# B&R Automation Studio project Soiled_PLC (part 8)

#### pr.st - Implementation code
```iecst
(********************************************************************
 * COPYRIGHT --
 ********************************************************************
 * Program: pr
 * File: pr.st
 * Author: treamsbottom
 * Created: July 16, 2015
 ********************************************************************
 * Implementation of program pr
 ********************************************************************)

PROGRAM _INIT
//Configuration
mySeq						:= 23;	//Sequence number
myIO						:= 11;
myZone						:= 0;
myRelLine					:= 31;
myBag						:= 243; //Buffer Bag
bufferSettleTime			:= 300;

myOutBag 					:= Line[myRelLine].LastBag;
END_PROGRAM

PROGRAM _CYCLIC
//Inputs
i_bagAtBuffer				:= X[myIO].X01;

i_bagAtBufferOut 		:= FALSE; // Any Single bag buffer out IO.
i_bufferOutOpen			:= FALSE;

o_openBuffer	:= FALSE;

IF (myBag = 0) THEN
	Alarm[mySeq].Bag	:= mySeq + 10000;
ELSE
	Alarm[mySeq].Bag	:= myBag;
END_IF;

Alarm[mySeq].Name 		:= 0;
Alarm[mySeq].Beacon		:= TRUE;
Alarm[mySeq].Extra		:= 0;
Alarm[mySeq].Time		:= 3000;

//Setup Sequence
step := D[900 + mySeq];
//Setup Pulse contact
pls := (step <> lastStep);
lastStep := step;

//Sequence
IF (step = 0) THEN
	//Disabled
END_IF;

//Bag Settled at buffer
ton_10ms_SettledBuffer(IN:= i_bagAtBuffer, PT:= bufferSettleTime);
IF (step = 1) THEN
	IF ton_10ms_SettledBuffer.Q AND NOT Std.HaltSysZone[myZone]THEN
		IF Line[myRelLine].Clear AND NOT i_bagAtBufferOut AND NOT i_bufferOutOpen AND NOT Line[myRelLine].Trip THEN
			IF (myBag = 0) THEN
				C[myRelLine] := 0;
				D[900 + mySeq] := 2;
			ELSIF (Bag[myBag].Cat > 0) AND (Bag[myOutBag].Cat = 0) THEN
				C[myRelLine] := 0;
				D[900 + mySeq] := 2;
			ELSIF (Bag[myBag].Cat = 0) THEN
				Alarm[mySeq].Name := ALM_BAG_DATA_ERROR;
				Alarm[mySeq].Time := 0;
			ELSIF (Bag[myOutBag].Cat > 0) THEN
				Alarm[mySeq].Name := ALM_BAG_DATA_ERROR;
				Alarm[mySeq].Bag := myOutBag;
				Alarm[mySeq].Time := 0;
			END_IF;
		ELSIF Line[myRelLine].Trip THEN
			Alarm[mySeq].Name := ALM_SWITCH_FAULT; //Trip is stuck on
			Alarm[mySeq].Time := 500;
		END_IF;
	ELSIF (myBag > 0) AND (Bag[myBag].Cat > 0) THEN
		Alarm[mySeq].Name := ALM_BAG_NOT_SETTLED;
	END_IF;
END_IF;

IF (step = 2) THEN
	dataValid := ((myBag = 0) OR ((Bag[myBag].Cat > 0) AND (Bag[myOutBag].Cat = 0)));
	o_openBuffer :=  dataValid;
	IF dataValid THEN
		IF Line[myRelLine].Trip THEN
			IF (myBag > 0) THEN
				Bag[myOutBag] := Bag[myBag];
				Bag[myBag]  := Bag[0];
			END_IF;
			D[900 + mySeq] := 1;
		END_IF;
		Alarm[mySeq].Name := ALM_BAG_NOT_RELEASED;
	ELSIF (myBag > 0) THEN
		IF (Bag[myBag].Cat = 0) THEN
			Alarm[mySeq].Name := ALM_BAG_DATA_ERROR;
			Alarm[mySeq].Time := 0;
		ELSIF (Bag[myOutBag].Cat > 0) THEN
			Alarm[mySeq].Name := ALM_BAG_DATA_ERROR;
			Alarm[mySeq].Bag := myOutBag;
			Alarm[mySeq].Time := 0;
		END_IF;
	END_IF;
END_IF;

//-----------------------------------
//PLC Outputs - adjust TO suit system
//-----------------------------------

Y[myIO].Y01 := o_openBuffer;

//Alarms
timerAlarm(IN := NOT pls AND (Alarm[mySeq].Name > 0),PT:= Alarm[mySeq].Time);

Alarm[mySeq].On 	:= timerAlarm.Q;
Alarm[mySeq].ET 	:= timerAlarm.ET;

END_PROGRAM
```

### Program Logical/Sequences/10ms/zzForceO (IEC)

#### zzforceo.ab
```automation-basic
;----------------------------
;Output forcing from Graphics
;----------------------------

;Version 1.00 02/09/2006 D.J. First Issue
;Version 2.00 20/11/2009 D.J. Changed to 8 I/O inputs per card

PROGRAM _INIT

;Clear force registers

D[380] = 0
D[381] = 0
D[382] = 0
D[383] = 0
D[384] = 0
D[385] = 0
D[386] = 0
D[386] = 0
D[387] = 0
D[388] = 0
D[389] = 0
D[390] = 0
D[391] = 0
D[392] = 0
D[393] = 0
D[394] = 0
D[395] = 0
D[396] = 0
D[396] = 0
D[397] = 0
D[398] = 0
D[399] = 0

;Clear force disable
memset(ADR(YForceDisable),0, SIZEOF(YForceDisable))

END_PROGRAM

PROGRAM _CYCLIC

LOOP Force = 1 TO 4 DO

	n = ((Force - 1) * 5)

	myForceCard 	= D[380 + n]
	myForceState 	= D[383 + n]
	myForceValue 	= D[384 + n]

	IF (myForceCard > Std.MaxIO) THEN
		myForceCard = 0
	ENDIF

	YForce.Y01 		= BIT_TST(myForceState,0)
	YForce.Y02 		= BIT_TST(myForceState,1)
	YForce.Y03 		= BIT_TST(myForceState,2)
	YForce.Y04 		= BIT_TST(myForceState,3)
	YForce.Y05 		= BIT_TST(myForceState,4)
	YForce.Y06 		= BIT_TST(myForceState,5)
	YForce.Y07 		= BIT_TST(myForceState,6)
	YForce.Y08 		= BIT_TST(myForceState,7)
	YForce.Y09 		= BIT_TST(myForceState,8)
	YForce.Y10 		= BIT_TST(myForceState,9)
	YForce.Y11 		= BIT_TST(myForceState,10)
	YForce.Y12 		= BIT_TST(myForceState,11)
	YForce.Y13 		= BIT_TST(myForceState,12)
	YForce.Y14 		= BIT_TST(myForceState,13)
	YForce.Y15 		= BIT_TST(myForceState,14)
	YForce.Y16 		= BIT_TST(myForceState,15)

	YForceVal.Y01 	= BIT_TST(myForceValue,0)
	YForceVal.Y02 	= BIT_TST(myForceValue,1)
	YForceVal.Y03 	= BIT_TST(myForceValue,2)
	YForceVal.Y04 	= BIT_TST(myForceValue,3)
	YForceVal.Y05 	= BIT_TST(myForceValue,4)
	YForceVal.Y06 	= BIT_TST(myForceValue,5)
	YForceVal.Y07 	= BIT_TST(myForceValue,6)
	YForceVal.Y08 	= BIT_TST(myForceValue,7)
	YForceVal.Y09 	= BIT_TST(myForceValue,8)
	YForceVal.Y10 	= BIT_TST(myForceValue,9)
	YForceVal.Y11 	= BIT_TST(myForceValue,10)
	YForceVal.Y12 	= BIT_TST(myForceValue,11)
	YForceVal.Y13 	= BIT_TST(myForceValue,12)
	YForceVal.Y14 	= BIT_TST(myForceValue,13)
	YForceVal.Y15 	= BIT_TST(myForceValue,14)
	YForceVal.Y16 	= BIT_TST(myForceValue,15)

	Y[myForceCard].Y01 = (Y[myForceCard].Y01 AND NOT YForce.Y01) OR (YForce.Y01 AND YForceVal.Y01)
	Y[myForceCard].Y02 = (Y[myForceCard].Y02 AND NOT YForce.Y02) OR (YForce.Y02 AND YForceVal.Y02)
	Y[myForceCard].Y03 = (Y[myForceCard].Y03 AND NOT YForce.Y03) OR (YForce.Y03 AND YForceVal.Y03)
	Y[myForceCard].Y04 = (Y[myForceCard].Y04 AND NOT YForce.Y04) OR (YForce.Y04 AND YForceVal.Y04)
	Y[myForceCard].Y05 = (Y[myForceCard].Y05 AND NOT YForce.Y05) OR (YForce.Y05 AND YForceVal.Y05)
	Y[myForceCard].Y06 = (Y[myForceCard].Y06 AND NOT YForce.Y06) OR (YForce.Y06 AND YForceVal.Y06)
	Y[myForceCard].Y07 = (Y[myForceCard].Y07 AND NOT YForce.Y07) OR (YForce.Y07 AND YForceVal.Y07)
	Y[myForceCard].Y08 = (Y[myForceCard].Y08 AND NOT YForce.Y08) OR (YForce.Y08 AND YForceVal.Y08)
	Y[myForceCard].Y09 = (Y[myForceCard].Y09 AND NOT YForce.Y09) OR (YForce.Y09 AND YForceVal.Y09)
	Y[myForceCard].Y10 = (Y[myForceCard].Y10 AND NOT YForce.Y10) OR (YForce.Y10 AND YForceVal.Y10)
	Y[myForceCard].Y11 = (Y[myForceCard].Y11 AND NOT YForce.Y11) OR (YForce.Y11 AND YForceVal.Y11)
	Y[myForceCard].Y12 = (Y[myForceCard].Y12 AND NOT YForce.Y12) OR (YForce.Y12 AND YForceVal.Y12)
	Y[myForceCard].Y13 = (Y[myForceCard].Y13 AND NOT YForce.Y13) OR (YForce.Y13 AND YForceVal.Y13)
	Y[myForceCard].Y14 = (Y[myForceCard].Y14 AND NOT YForce.Y14) OR (YForce.Y14 AND YForceVal.Y14)
	Y[myForceCard].Y15 = (Y[myForceCard].Y15 AND NOT YForce.Y15) OR (YForce.Y15 AND YForceVal.Y15)
	Y[myForceCard].Y16 = (Y[myForceCard].Y16 AND NOT YForce.Y16) OR (YForce.Y16 AND YForceVal.Y16)

ENDLOOP

END_PROGRAM
```

### Program Logical/Sequences/10ms/zzStnSer (IEC, version 3.00.1)

#### zzstnser.var
```iecst
VAR
	MixProgTyp : BOOL;
	BatchFound : BOOL;
	MixCusts : BOOL;
	MixProgs : BOOL;
	MatchCust : BOOL;
	MatchBags : BOOL;
	MatchProgType : BOOL;
	MatchProg : BOOL;
	MatchCat : BOOL;
	StartPurge : BOOL;
	MixCats : BOOL;
	BankValid : BOOL;
	LineValid : BOOL;
	BagInList : ARRAY[0..30] OF BOOL;
	StartPurgeET : UDINT;
	BagNum : UINT;
	BagWgt : UINT;
	Index : UINT;
	PurgeBagsQty : UINT;
	StnNum : UINT;
	BatchCount : UINT;
	s : UINT;
	BatchWeight : UINT;
	myBag : UINT;
	r : UINT;
	MaxReverseWeight : UINT;
END_VAR
VAR RETAIN
	LineSearchManual : UINT;
END_VAR
VAR
	NumberOfPurgeBags : UINT;
	x : UINT;
END_VAR
VAR RETAIN
	SearchLine : UINT;
END_VAR
VAR
	Bank : UINT;
	Choice : UINT;
	EndofBagArray : UINT;
	PurgeBatchSize : UINT;
	MaxBatchWieght : UINT;
END_VAR
VAR RETAIN
	n : UINT;
END_VAR
VAR
	t : UINT;
	myBag_x : UINT;
	myBag_n : UINT;
END_VAR
VAR RETAIN
	SearchFound : UINT;
END_VAR
VAR
	LineSearch : ARRAY[0..4] OF UINT;
	SearchBagArray : ARRAY[0..30] OF UINT;
	PurgeBags : ARRAY[0..30] OF UINT;
	PurgeBagsInWgtOrder : ARRAY[0..30] OF UINT;
	PurgeOn : UINT;
	StatusReg : ARRAY[0..1] OF UDINT;
	SearchIndex : USINT;
	ReSearch : BOOL;
	MisMatchedLoad : BOOL;
	y : INT;
	Break : BOOL;
	StnCat : UDINT;
	GetStn : UINT;
	TestTim : BOOL;
	myStartStop : UINT;
	b : UINT;
	TON_Purge : ARRAY[0..4] OF TON_10ms;
	myBatchWgt : UDINT;
	test : UDINT;
	TEST : BOOL;
END_VAR
```

#### zzstnser.ab
```automation-basic
;-----------------------------------------------------
;Sorting Station Search Routine - No changes required!
;-----------------------------------------------------

;----------------------------------------
;Version 1.00 19/12/2005 First Issue D.J.
;Version 2.00 03/11/2010 Revised D.J.
;Version 3.00 19/07/2016 TR... Fix bug so multiple banks can release whilst purging..
;----------------------------------------

PROGRAM _CYCLIC

;Only one Bank / Loading VC can search in a given scan.

myStartStop			= 100 ; Start of Start Stops

IF myStartStop >= 100 THEN
	myStartStop = myStartStop + 7600
ENDIF

Bank = Bank + 1
IF (Bank > Std.MaxStationBanks) THEN
	Bank = 1
ENDIF
;Clear arrays
LOOP n = 0 TO Std.MaxWeighstations DO
	BagInList[n] = FALSE
	SearchBagArray[n] = 0
ENDLOOP

;Clear Array
LOOP b = 1 TO 4 DO
	Std.StnsToPurge[b] = FALSE
	LOOP n = 1 TO Ldg[b].NoStations DO
		x = Ldg[b].Stations[n]
		IF Stn[x].Purge THEN
			Std.StnsToPurge[b] = TRUE
		ENDIF
	ENDLOOP
	TON_Purge[b].IN = Std.StnsToPurge[b]
	TON_Purge[b].PT = 100
	TON_Purge[b] FUB TON_10ms()
	//TON_10ms(Std.StnsToPurge,100,StartPurge,StartPurgeET) ; use a timer to wait for all purge events to be recieved from trackview
ENDLOOP

MixCats			= (D[369] > 0)
MixCusts		= (D[366] > 0)	;Allow mixing of customers?
MixProgs		= (D[367] > 0)	;Allow mixing of Programs?
MixProgTyp		= (D[368] > 0) 	;Allow mixing of Program Types?

;Mix Options are enforced in Trackview - If we do it in the PLC we cannot turn off Mixing.
;IF MixProgTyp THEN
;	D[367] = 1 //Mix Progs
;	D[369] = 1 //Mix Cats
;ELSE IF MixProgs THEN					;IF mixing programs then category must be mixed also.....
;	D[369] =  1 // Mix Cats
;ENDIF

;IF Std.ReversingBelt THEN
	MaxReverseWeight	= D[370]			;Max weight to reverse..
;ELSE
;	MaxReverseWeight = 0
;ENDIF
;Send Status to Trackview -- BitWise OR to look at all banks

PurgeOn = (Std.PurgeBank[1].PurgeOn OR Std.PurgeBank[2].PurgeOn OR Std.PurgeBank[3].PurgeOn OR Std.PurgeBank[4].PurgeOn)
StatusReg[0] = (Std.PurgeBank[1].StationsStatus[0] OR Std.PurgeBank[2].StationsStatus[0] OR Std.PurgeBank[3].StationsStatus[0] OR Std.PurgeBank[4].StationsStatus[0])
StatusReg[1] = (Std.PurgeBank[1].StationsStatus[1] OR Std.PurgeBank[2].StationsStatus[1] OR Std.PurgeBank[3].StationsStatus[1] OR Std.PurgeBank[4].StationsStatus[1])
D[360] = PurgeOn
memcpy(ADR(D[371]),ADR(StatusReg),4)
;Used by other sequences that need to check for Line[x].SpaceBIT direct
;eg. Loading VC will look for Enable.Search = 3
Enable.Search = Bank

IF (Bank <= Std.MaxStationBanks) THEN

	IF (Ldg[Bank].Search = 1) THEN
		StartPurge = TON_Purge[Bank].Q
		Ldg[Bank].Found = 0
		Ldg[Bank].Line  = 0

		SearchFound = 0
		SearchLine  = 0

		Stn[0].QTime = 0

		LOOP x = 1 TO Ldg[Bank].NoStations DO
			n = Ldg[Bank].Stations[x]
			IF (Std.StnsToPurge[Bank] AND Std.AutoPurge) THEN	;Search through purge Stations to find bags that can be mixed

				IF Bank = 1 THEN
					Break
;					IF NOT TestTim THEN
;						GOTO Debug
;					ENDIF
				ELSE IF Bank = 2 THEN
					Break
				ENDIF
				;Purge doesn;t need to be in x loop so exit if > 1
				EXITIF x > 1
				IF StartPurge THEN
					PurgeBatchSize	= 0
					BatchFound = FALSE
					; 1st put all bags to be searched into an array to reduce scanning through all stations bags
					//LOOP r = 0 TO Std.MaxWeighstations DO
					LOOP r = 1 TO Ldg[Bank].NoStations DO
						Std.PurgeBank[Bank].PurgeBatch[r] = 0
						n = Ldg[Bank].Stations[r]
						IF Stn[n].Purge AND (Stn[n].Weight > 0) AND NOT BagInList[n] THEN //AND (r >= Ldg[Bank].StartStn) AND (r <= Ldg[Bank].EndStn)  THEN
							SearchBagArray[Ldg[Bank].NoStations] = LDG_GetBagFromStation(Std.StationBagsStart,n)
							BagInList[n] = TRUE
						ENDIF
						;Shuffle array
						LOOP s = Ldg[Bank].NoStations DOWNTO 1 DO
							IF (SearchBagArray[s-1] = 0) AND (SearchBagArray[s] > 0) THEN
								SearchBagArray[s-1] = SearchBagArray[s]
								SearchBagArray[s] = 0
								EndofBagArray = (s - 1)
							ENDIF
						ENDLOOP
					ENDLOOP
					;LOOP r = 0 TO EndofBagArray DO ; Start Searching through bags
					r = 0 ;Only search through from 1st bag in array as we already know it is to purge
					ReSearch = FALSE
					MisMatchedLoad = FALSE
					SearchIndex = 0
					StartSearch: ;Marker to re-search
					IF ReSearch THEN
						r = SearchIndex
					ENDIF
					LOOP s = 0 TO Std.MaxWeighstations DO
						PurgeBags[s] = 0
					ENDLOOP
					LOOP s = EndofBagArray DOWNTO 0 DO
						myBag_n = SearchBagArray[r]
						myBag_x = SearchBagArray[s]
						MatchCust = FALSE
						MatchCat = FALSE
						MatchProgType = FALSE
						MatchProg = FALSE
						BankValid = TRUE;((myBag_n >= Ldg[Bank].StartStn) AND (myBag_n <= Ldg[Bank].EndStn) AND (myBag_x >= Ldg[Bank].StartStn) AND (myBag_x <= Ldg[0].EndStn))

						;Check customer 1st
						IF (Bag[myBag_n].Cus = Bag[myBag_x].Cus) OR MixCusts THEN
							MatchCust = TRUE
						ENDIF
						IF (Bag[myBag_n].Cat = Bag[myBag_x].Cat) OR MixCats THEN
							MatchCat = TRUE
						ENDIF
						IF (Bag[myBag_n].Prg = Bag[myBag_x].Prg) OR MixProgs THEN
							MatchProg = TRUE
						ENDIF
						IF (D[2900 + Bag[myBag_n].Prg] = D[2900 + Bag[myBag_x].Prg]) OR MixProgTyp THEN
							MatchProgType = TRUE
						ENDIF

						MatchBags = (MatchCust AND MatchCat AND MatchProg AND MatchProgType AND BankValid)
						IF MatchBags THEN ; Put bag into another array so they can be best matched by weight
							;PurgeBags[0] = myBag_n
							PurgeBags[Std.MaxWeighstations] = myBag_x
							LOOP t = Std.MaxWeighstations DOWNTO 1 DO
								IF (PurgeBags[t] > 0) AND (PurgeBags[t-1] = 0) THEN
									PurgeBags[t -1] = PurgeBags[t]
									PurgeBags[t] = 0
									PurgeBatchSize	= t
								ENDIF
							ENDLOOP
						ENDIF
					ENDLOOP ; Ony research if no matching bags, and the bag searched is to small for a batch
					//Get Total weight of batch to see if matched bags meet minumum weight criteria.
					myBatchWgt = 0
					LOOP t = 0 TO PurgeBatchSize DO
						myBatchWgt = myBatchWgt + Bag[PurgeBags[t]].Wgt
					ENDLOOP
					//IF ((PurgeBatchSize = 1) AND (Bag[PurgeBags[0]].Wgt < MaxReverseWeight)) THEN
					IF ((PurgeBatchSize >= 1) AND (myBatchWgt < MaxReverseWeight)) THEN
						ReSearch = TRUE
						INC SearchIndex
						;Check when all bags have been searched...
						IF (SearchBagArray[SearchIndex] = 0) THEN
							;INC SearchIndex
							;The only bags left cannot be put in the same bag and should be classified as a mixed load.
							MisMatchedLoad = (SearchIndex > 1)
							LOOP y = 0 TO SearchIndex - 1 DO
								PurgeBags[y] = 	SearchBagArray[y]
							ENDLOOP
							PurgeBatchSize = SearchIndex
						ELSE
							GOTO StartSearch
						ENDIF
					ENDIF

					;ENDLOOP
					;Matching bags are in the array Purge Bags. Try to fit into a load?
					;Bag 0 in the array is that master.. This is the data that will go into a bag.. so we will get the batch weight from this program code.
					;Put all bag into wieght order highest first..
					LOOP r = 0 TO 30 DO
						BagInList[r] = FALSE
						PurgeBagsInWgtOrder[r] = 0
					ENDLOOP

					IF (PurgeBatchSize > 0) THEN
						//Find the lowest SP3 from all bag in the purge array...
						MaxBatchWieght = 0
						LOOP r = 0 TO ((SIZEOF(PurgeBags)/SIZEOF(PurgeBags[0])) - 1) DO
							EXITIF PurgeBags[r] = 0
							GetStn =  (PurgeBags[r] - Std.StationBagsStart + 1)
							IF (GetStn <= Std.MaxWeighstations) AND (D[4900 + GetStn] > 0) AND ((MaxBatchWieght > D[4900 + GetStn]) OR (MaxBatchWieght = 0))    THEN
								MaxBatchWieght = D[4900 + GetStn] ;SP3
							ENDIF
						ENDLOOP

						IF (MaxBatchWieght = 0) OR (MaxBatchWieght <= MaxReverseWeight) THEN
							 MaxBatchWieght = MaxReverseWeight + 100
						ENDIF

						LOOP r = 0 TO (PurgeBatchSize - 1) DO
							BagWgt = 0
							LOOP s = 0 TO (PurgeBatchSize - 1) DO
								IF (Bag[PurgeBags[s]].Wgt > 0) AND (Bag[PurgeBags[s]].Wgt > BagWgt) AND NOT BagInList[s] THEN
									BagWgt = Bag[PurgeBags[s]].Wgt
									BagNum = PurgeBags[s]
									Index = s
								ENDIF
							ENDLOOP
							PurgeBagsInWgtOrder[r] = BagNum
							BagInList[Index] = TRUE
						ENDLOOP ;
						IF (MaxBatchWieght > MaxReverseWeight) AND (Bag[PurgeBagsInWgtOrder[0]].Wgt > 0)THEN ; Check no errors in batch sizes.. Reverse all loads if fault
							;Now bags are in weight order make the best by adding the highest values until bag is full
							BatchWeight = 0
							PurgeBagsQty = 0
							;IF (Bag[PurgeBagsInWgtOrder[0]].Wgt  < MaxBatchWieght) THEN
							BatchWeight = Bag[PurgeBagsInWgtOrder[0]].Wgt
							BatchCount = Bag[PurgeBagsInWgtOrder[0]].Cnt
							Std.PurgeBank[Bank].PurgeBatch[0] = PurgeBagsInWgtOrder[0]
							;ENDIF
							LOOP r = 1 TO PurgeBatchSize DO ; Start from 1 as index 0 is highest weight so always in the array
								myBag = PurgeBagsInWgtOrder[r]
								IF ((Bag[myBag].Wgt + BatchWeight) <= MaxBatchWieght) THEN
									BatchWeight = Bag[myBag].Wgt + BatchWeight
									BatchCount = Bag[myBag].Cnt + BatchCount
									Std.PurgeBank[Bank].PurgeBatch[PurgeBatchSize] = myBag
									PurgeBagsQty = PurgeBagsQty + 1
								ENDIF
								;Shuffle down array
								LOOP s = PurgeBatchSize DOWNTO 1 DO
									IF (Std.PurgeBank[Bank].PurgeBatch[s] > 0) AND (Std.PurgeBank[Bank].PurgeBatch[s - 1] = 0) THEN
										Std.PurgeBank[Bank].PurgeBatch[s - 1] = Std.PurgeBank[Bank].PurgeBatch[s]
										Std.PurgeBank[Bank].PurgeBatch[s] = 0
									ENDIF
								ENDLOOP
								IF (r = PurgeBatchSize) AND (Std.PurgeBank[Bank].PurgeBatch[0] > 0) THEN
									BatchFound = TRUE
								ENDIF
							EXITIF BatchFound = TRUE
							ENDLOOP
						ENDIF
;					ELSE
;						GOTO ExitPurge ;Invalid purge..
					ENDIF
					IF BatchFound AND NOT MisMatchedLoad THEN ;Bags found;
						IF (BatchWeight >=  MaxReverseWeight) THEN ; Wieght it OK purge into Bag search for destination.

							IF Std.AutoLineAllocation THEN
								SearchFound  		= 99
								SearchLine   		= 0;LineSearch[Choice]
								Ldg[Bank].Search   	= 2
							ELSE	;
								;Check line choice 1st to 4th in order if any valid then exit loop
								;StnNum = (Std.PurgeBank[Bank].PurgeBatch[0] - (Std.StationBagsStart[Bank] - Ldg[Bank].StartStn)) ; Get station number from Bag number.
								StnCat =  Bag[Std.PurgeBank[Bank].PurgeBatch[0]].Prg

								LineSearch[1]   = D[3000 + StnCat]
								LineSearch[2]   = D[3100 + StnCat]
								LineSearch[3]   = D[3200 + StnCat]
								LineSearch[4]   = D[3300 + StnCat]

								LOOP Choice = 1 TO 4 DO
									LineValid = (D[myStartStop + LineSearch[Choice]] > 0)
									IF (LineSearch[Choice] > 0) AND (Line[LineSearch[Choice]].SpaceBIT >= 1) AND LineValid THEN
										SearchFound  		= 99
										SearchLine   		= LineSearch[Choice]
										Ldg[Bank].Search   	= 2
									ENDIF
									EXITIF (SearchFound > 0)
								ENDLOOP
							ENDIF
						ELSE ; Load/s is to small reverse.

							SearchFound  		= 98
							SearchLine   		= 0
							Ldg[Bank].Search   	= 2
						ENDIF
					ELSE IF MisMatchedLoad THEN
						SearchFound  		= 97
						SearchLine   		= 0
						Ldg[Bank].Search   	= 2
					ENDIF
					IF SearchFound > 90 THEN ;If bags are found remove from purging Q
						Std.PurgeBank[Bank].PurgeBagQty	= PurgeBagsQty

						Std.PurgeBank[Bank].PurgeBatchWieght = BatchWeight
						Std.PurgeBank[Bank].PurgeBatchCount	= BatchCount
;						LOOP r = 0 TO PurgeBagsQty - 1 DO
;							IF (Std.PurgeBank[Bank].PurgeBatch[r] > 0) THEN
;								StnNum = (Std.PurgeBank[Bank].PurgeBatch[r] - (Std.StationBagsStart[Bank] - Ldg[Bank].StartStn))
;								;Stn[StnNum].QTime = 0
;								;Stn[StnNum].Purge = FALSE
;							ENDIF
;						ENDLOOP
					ENDIF
				ENDIF
			ELSE IF ((Stn[n].QTime > 10) AND (Stn[n].QTime > Stn[0].QTime)) OR (TEST) THEN

				;Destination has been given to bag by operator check
				LineSearchManual = Stn[n].DestManual

				IF Std.AutoLineAllocation THEN

					;Automatic Line Allocation - Line Space is never checked even if a destiantion has been edited
					SearchFound  		= n
					SearchLine   		= LineSearchManual
					Stn[0].QTime 		= Stn[n].QTime
					Ldg[Bank].Search   	= 2

				ELSE
					;1st 2nd 3rd and 4th Line choices
					LineSearch[1]   = D[4000 + n]
					LineSearch[2]   = D[4100 + n]
					LineSearch[3]   = D[4200 + n]
					LineSearch[4]   = D[4300 + n]

					;Always Search for at least 1 space
					IF (Stn[n].SpacesRequired = 0) THEN
						Stn[n].SpacesRequired = 1
					ENDIF

					;When manual is selected then the 1st 2nd 3rd and 4th are not checked
					IF (LineSearchManual > 0) THEN
						IF (Line[LineSearchManual].SpaceBIT > 0) THEN
							SearchFound  		= n
							SearchLine   		= LineSearchManual
							Stn[0].QTime 		= Stn[n].QTime
							Ldg[Bank].Search   	= 2
						ENDIF
					ELSE
							;Check line choice 1st to 4th in order if any valid then exit loop

						LOOP Choice = 1 TO 4 DO
							;Choice = 1
							LineValid = (D[myStartStop + LineSearch[Choice]] > 0)
							IF (LineSearch[Choice] > 0) AND (LineSearch[Choice] < 7) AND (Line[LineSearch[Choice]].SpaceBIT >= Stn[n].SpacesRequired) AND LineValid THEN
								SearchFound  		= n
								SearchLine   		= LineSearch[Choice]
								Stn[0].QTime 		= Stn[n].QTime
								Ldg[Bank].Search   	= 2

							ENDIF
							EXITIF (SearchFound > 0)

							IF (LineSearch[Choice] > 13) AND (D[LineSearch[Choice]]>0) THEN
								IF (Line[9].SpaceBIT > 0) THEN
									SearchFound  		= n
									SearchLine   		= LineSearch[Choice]
									Stn[0].QTime 		= Stn[n].QTime
									Ldg[Bank].Search   	= 2
								ENDIF
							ENDIF

						ENDLOOP

					ENDIF

				ENDIF ;/AutoLineAllocation

			ENDIF

		ENDLOOP

		ExitPurge:
		IF (Ldg[Bank].Search = 2) THEN
			Ldg[Bank].Found  = SearchFound
			Ldg[Bank].Line   = SearchLine
		ELSE
			Ldg[Bank].Search = 0 ;Failed
		ENDIF

	ENDIF
ENDIF
Debug:

END_PROGRAM
```

### Program Logical/Sequences/10ms/zzStatus (IEC) - * System status

#### zzstatus.var
```iecst
VAR
	OngoingStopped : BOOL;
	OffgoingStopped : BOOL;
	LoadingStopped : BOOL;
	tmrForce : TON_10ms;
	ForceEnable : BOOL;
	tmrBeltPLS_A : TON_10ms;
	A_PT : UDINT;
	tmrBeltPLS_B : TON_10ms;
	B_PT : UDINT;
	CarouselPhotocell : BOOL;
	tmrCaroPhotoClear : TON_10ms;
	CaroClearPT : UDINT;
	RunSB10 : BOOL;
	tmrCaroPhotoBlocked : TON_10ms;
	CaroBlockedPT : UDINT;
	tmrClearSDC3 : TON_10ms;
	SDC3BagOpen : BOOL;
	ForceBelt : BOOL;
	RunSB11 : BOOL;
	SB10Photocell : BOOL;
	SB11Photocell : BOOL;
	tmrSB11Clear : TON_10ms;
	tmrSB10Clear : TON_10ms;
	tmrBeltPLS_C : TON_10ms;
	tmrBeltPLS_D : TON_10ms;
	C_PT : UDINT;
	D_PT : UDINT;
	I_EndOfBelt : BOOL;
	O_Run : BOOL;
	I_SelectAuto : BOOL;
	MaxZones : UINT;
	n : UINT;
	TEST : BOOL;
END_VAR
```

#### zzstatus.ab
```automation-basic
PROGRAM _CYCLIC
(* cyclic program *)

;System Status and Halting
;-------------------------

Std.StopSystem 				= (D[100] <> 0)

;Std.EStop 					= NOT X[3].X01
;Std.MotorOverload   		= X[3].X01 AND NOT X[3].X03
;Std.SafetyOn				= X[6].X16
;Std.HaltSys 				= NOT Std.SafetyOn ;OR Std.StopSystem)
;
;;Std.SafetyHighLevel			= TRUE

;MaxZones = 4
;Std.SafetyOnZone[0]			= Std.SafetyOn
;Std.SafetyOnZone[1]			= FALSE;Guarded area
;Std.SafetyOnZone[2]			= FALSE
;Std.SafetyOnZone[3]			= FALSE
;Std.SafetyOnZone[4]			= FALSE
;
;LOOP n = 0 TO MaxZones DO
;	Std.HaltSysZone[n] =  NOT Std.SafetyOnZone[n]

;ENDLOOP
Std.EStop 					= NOT X[11].X16

Std.MotorOverload   		= X[9].X15 AND NOT X[9].X16
Std.SafetyOn				=  X[11].X16 ;X[6].X16 OR TestSystem ;(SafetyZone[0].Zone_Status AND NOT SafetyZone[0].Disable) OR TestSystem;
Std.HaltSys					= NOT Std.SafetyOn OR TEST
Std.HaltSysZone[0]	        = Std.HaltSys
LOOP n = 0 TO MAX_SAFE_ZONES DO
;	Std.SafetyOnZone[n]	= (SafetyZone[n].Zone_Status AND NOT SafetyZone[n].Disable) OR TestSystem;
;	Std.HaltSysZone[n] =  NOT Std.SafetyOnZone[n]
ENDLOOP

;set to TRUE if not required
LoadingStopped 	= TRUE ;(Bag[220].Prg = 0)
OngoingStopped 	= TRUE ;(Bag[224].Prg = 0)
OffgoingStopped = TRUE ;(Bag[225].Prg = 0)

;If no Bag In Transit and stop requested then set system to stopped D[100] = 2
IF Std.StopSystem THEN
	IF LoadingStopped AND OngoingStopped AND OffgoingStopped THEN
		D[100] = 2
	ENDIF
ENDIF

;Force I/O Enable - Max ? Minutes
ForceEnable = FALSE

tmrForce.IN = ForceEnable
tmrForce.PT = 90000 ;6000 = 1 Minute
tmrForce FUB TON_10ms()

IF ForceEnable AND NOT tmrForce.Q THEN
	D[319] = 1
ELSE
	D[319] = 0
ENDIF

END_PROGRAM
```

- Program Logical/Sequences/10ms/zzIndi (IEC) - * Indication pictures on graphics (no source held here)

### Program Logical/Sequences/10ms/zzTCPIP (IEC, version 5.00.0) - * TCP IP Communications For Driver V5.0 and above

#### zztcpip.ab
```automation-basic
;-----------------------------------
;TCP IP Driver Communications Driver
;-----------------------------------

;------------------------------------------------------------------------------------------------------------
;Version 1.00 01/12/2005 D.J. First Issue
;Version 2.00 14/04/2009 D.J. Added VC_Posn data type
;Version 3.00 02/06/2009 D.J. Added D32 32-Bit Data
;Version 4.00 09/04/2010 D.J. Added MCN Machine Type Communication
;Version 4.10 03/11/2010 D.J. Changed VC to RB (Robo) other than that full compatiable with Version 4.00
;Version 5.00 28/04/2012 D.J. Enabled larger data size now 5000 bytes (200 bags with a size of 25 bytes each)
;------------------------------------------------------------------------------------------------------------

;Normally the driver will be sending constant requests - if the driver dosen't send anything for 1 second then the connection should be closed.

PROGRAM _INIT

;Enable connections set to TRUE or FALSE depending on how many connections are required
EnableConnection1 = TRUE
EnableConnection2 = TRUE

;Start Connection
ResetConnection = TRUE

END_PROGRAM

PROGRAM _CYCLIC

;------------
;Connection 1
;------------

;Restart - from init routine
IF ResetConnection THEN
	IF EnableConnection1 THEN
		NEWSTEP = 1
	ELSE
		NEWSTEP = 0
	ENDIF
ENDIF

STEP = NEWSTEP

;Disabled
IF STEP = 0 THEN
	;Do Nothing
ENDIF

;Init Server
IF STEP = 1 THEN
	TCPserv_1.enable = 1
	TCPserv_1.porta = 21001
	TCPserv_1 FUB TCPserv()
	IPAddr	= H_TO_NUDINT(TCPserv_1.ipaddr)
	Port	= TCPserv_1.portb
	NEWSTEP = 2
ENDIF

;Server to listening - until PC connects
IF STEP = 2 THEN
	TCPserv_1 FUB TCPserv()
	IPAddr	= H_TO_NUDINT(TCPserv_1.ipaddr)
	Port	= TCPserv_1.portb
	IF TCPserv_1.status = 0 THEN
		PLS = TRUE
		NEWSTEP = 3
	ELSE IF TCPserv_1.status = 27155 THEN 							;27155 = No buffer space available
		NEWSTEP = 6
	ENDIF
ENDIF

;PC Connected - if error then disconnect
IF STEP = 3 THEN

	WriteEnable = FALSE

	IF TCPsend_1.status = 0 THEN

		TCPrecv_1.enable = 1
		TCPrecv_1.cident = TCPserv_1.cident
		TCPrecv_1.buffer = ADR(rdata[0])
		TCPrecv_1.mxbuflng = SIZEOF(rdata)
		TCPrecv_1 FUB TCPrecv()
		RXLength = TCPrecv_1.rxbuflng
		RXStatus = TCPrecv_1.status

		IF RXLength > 0 THEN

			Data_RXTX_Type  = rdata[1] 								;WR = 1  WW = 3
			Data_Array_Type = rdata[2]								;C  = 1 D  = 2 Bag = 3

			Data_StartH = rdata[3]
			Data_Start 	= LSL(Data_StartH,8) + rdata[4]
			Data_AmountH = rdata[5]
			Data_Amount = LSL(Data_AmountH,8) + rdata[6]

			IF Data_Array_Type = 1 THEN
				Data_array_adr 	= pC
				Bytes			= 2
			ELSE IF Data_Array_Type = 2 THEN
				Data_array_adr = pD
				Bytes			= 2
			ELSE IF Data_Array_Type = 3 THEN
				Data_array_adr 	= pBag
				Bytes			= SIZEOF(Bag[0])
			ELSE IF Data_Array_Type = 4 THEN
				Data_array_adr 	= pRB_Posn
				Bytes			= SIZEOF(RB_Posn[0])
			ELSE IF Data_Array_Type = 5 THEN
				Data_array_adr 	= pD32
				Bytes			= SIZEOF(D32[0])
			ELSE IF Data_Array_Type = 6 THEN
				Data_array_adr 	= pMCN
				Bytes			= SIZEOF(MCN[0])
			ENDIF

			PacketID = rdata[RXLength - 1] ;Packet ID sent back to Driver for check

			;Increase tx_frame and rx frame now 5000 bytes (Data_Amount based on 16 bit register 2 bytes)
			Data_Valid = ((Data_RXTX_Type > 0) AND (Data_Array_Type > 0) AND (Data_array_adr > 0) AND (Data_Amount > 0) AND (Data_Amount <= 2500))

			IF Data_Valid THEN

				RXValid = RXValid + 1

				IF (Data_RXTX_Type = 1) THEN					;Word Read - Transmit Data to PC

					tx_frame[0] = rdata[0]						;PLC Station

					memcpy(adr(tx_frame[1]),Data_array_adr + (Data_Start * Bytes),(Data_Amount * Bytes))

					tx_frame[(Data_Amount * Bytes) + 1] = PacketID ;USINT(0) ;Checksum not required
					tx_length 	= (Data_Amount * Bytes) + 2
					WriteEnable = TRUE

				ELSE IF (Data_RXTX_Type = 3) THEN 				;Word Write - Receive data from PC

					LengthValid = (RXLength > (Data_Amount * Bytes))
					IF LengthValid THEN
						memcpy(Data_array_adr + (Data_Start * Bytes),adr(rdata[7]),(Data_Amount * Bytes))

						tx_frame[0] = $06							;ACK
						tx_frame[1] = rdata[0]						;PLC Station
						tx_length 	= 2
						WriteEnable	= TRUE							;Set write enable
					ELSE
						tx_frame[0] = $15 							;NAK
						tx_frame[1] = rdata[0] 						;PLC Station
						tx_length 	= 2
						WriteEnable	= TRUE							;Set write enable

					ENDIF

				ENDIF

			ELSE

				tx_frame[0] = $15 								;NAK
				tx_frame[1] = rdata[0] 							;PLC Station
				tx_length 	= 2
				WriteEnable	= TRUE								;Set write enable

			ENDIF

			IF WriteEnable THEN
				TCPsend_1.enable = 1
    			TCPsend_1.cident = TCPserv_1.cident
    			TCPsend_1.buffer = ADR(tx_frame[0])
    			TCPsend_1.buflng = tx_length ;SIZEOF(tx_frame)
    			TCPsend_1 FUB TCPsend()
	    	ENDIF

	    ENDIF

	ELSE
		TCPsend_1 FUB TCPsend()
	ENDIF

    IF (((TCPsend_1.status <> 0) AND (TCPsend_1.status <> 65535)) OR NoData) THEN
    	NoData  = FALSE
    	NEWSTEP = 4
    ENDIF

ENDIF
TON_10ms(((STEP = 3) AND (RXLength = 0)),500,NoData,NoDataET)

;Close the connection - if closed then go-to listen else go-to wait for close
IF STEP = 4 THEN
	TCPclose_1.enable = 1
	TCPclose_1.cident = TCPserv_1.cident
	TCPclose_1 FUB TCPclose()
	NEWSTEP = 5
ENDIF

;Closing - wait until connection closed
IF STEP = 5 THEN
	IF TCPclose_1.status <> 0 THEN
		TCPclose_1 FUB TCPclose()
	ELSE IF TCPclose_1.status = 0 THEN
		TCPsend_1.status = 0
		NEWSTEP = 1
	ENDIF
ENDIF

IF STEP = 6 THEN
	;Warm / Cold Start Required
ENDIF

;------------
;Connection 2
;------------

;Restart - from init routine
IF ResetConnection THEN
	IF EnableConnection2 THEN
		NEWSTEP2 = 1
	ELSE
		NEWSTEP2 = 0
	ENDIF
ENDIF

STEP2 = NEWSTEP2

;Disabled
IF STEP2 = 0 THEN
	;Do Nothing
ENDIF

;Init Server
IF STEP2 = 1 THEN
	TCPserv_2.enable = 1
	TCPserv_2.porta = 21002
	TCPserv_2 FUB TCPserv()
	IPAddr2	= H_TO_NUDINT(TCPserv_2.ipaddr)
	Port2	= TCPserv_2.portb
	NEWSTEP2 = 2
ENDIF

;Server to listening - until PC connects
IF STEP2 = 2 THEN
	TCPserv_2 FUB TCPserv()
	IPAddr2	= H_TO_NUDINT(TCPserv_2.ipaddr)
	Port2	= TCPserv_2.portb
	IF TCPserv_2.status = 0 THEN
		PLS2 = TRUE
		NEWSTEP2 = 3
	ELSE IF TCPserv_2.status = 27155 THEN								;27155 = No buffer space available
		NEWSTEP2 = 6
	ENDIF
ENDIF

;PC Connected - if error then disconnect
IF STEP2 = 3 THEN

	WriteEnable2 = FALSE

	IF TCPsend_2.status = 0 THEN

		TCPrecv_2.enable = 1
		TCPrecv_2.cident = TCPserv_2.cident
		TCPrecv_2.buffer = ADR(rdata2[0])
		TCPrecv_2.mxbuflng = SIZEOF(rdata2)
		TCPrecv_2 FUB TCPrecv()
		RXLength2 = TCPrecv_2.rxbuflng
		RXStatus2 = TCPrecv_2.status

		IF RXLength2 > 0 THEN

			Data_RXTX_Type  = rdata2[1] 								;WR = 1 BR = 2 WW = 3 BW = 4 - Bit Read and Bit Write not used
			Data_Array_Type = rdata2[2]									;C  = 1 D  = 2 E  = 3

			Data_StartH = rdata2[3]
			Data_Start 	= LSL(Data_StartH,8) + rdata2[4]
			Data_AmountH = rdata2[5]
			Data_Amount = LSL(Data_AmountH,8) + rdata2[6]

				IF Data_Array_Type = 1 THEN
				Data_array_adr 	= pC
				Bytes			= 2
			ELSE IF Data_Array_Type = 2 THEN
				Data_array_adr = pD
				Bytes			= 2
			ELSE IF Data_Array_Type = 3 THEN
				Data_array_adr 	= pBag
				Bytes			= SIZEOF(Bag[0])
			ELSE IF Data_Array_Type = 4 THEN
				Data_array_adr 	= pRB_Posn
				Bytes			= SIZEOF(RB_Posn[0])
			ELSE IF Data_Array_Type = 5 THEN
				Data_array_adr 	= pD32
				Bytes			= SIZEOF(D32[0])
			ELSE IF Data_Array_Type = 6 THEN
				Data_array_adr 	= pMCN
				Bytes			= SIZEOF(MCN[0])
			ENDIF

			PacketID = rdata2[RXLength2 - 1] ;Packet ID sent back to Driver for check

			Data_Valid = ((Data_RXTX_Type > 0) AND (Data_Array_Type > 0) AND (Data_array_adr > 0) AND (Data_Amount > 0) AND (Data_Amount < 1001))

			IF Data_Valid THEN

				RXValid2 = RXValid2 + 1

				IF (Data_RXTX_Type = 1) THEN							;Word Read - Transmit Data to PC

					tx_frame2[0] = rdata2[0] 							;PLC Station

					memcpy(adr(tx_frame2[1]),Data_array_adr + (Data_Start * Bytes),(Data_Amount * Bytes))

					tx_frame2[(Data_Amount * Bytes) + 1] = PacketID ;USINT(0) ;Checksum not required
					tx_length2 	= (Data_Amount * Bytes) + 2
					WriteEnable2 = TRUE

				ELSE IF (Data_RXTX_Type = 3) THEN 						;Word Write - Receive data from PC

					LengthValid = (RXLength2 > (Data_Amount * Bytes))
					IF LengthValid THEN
						memcpy(Data_array_adr + (Data_Start * Bytes),adr(rdata2[7]),(Data_Amount * Bytes))

						tx_frame2[0] = $06									;ACK
						tx_frame2[1] = rdata2[0] 							;PLC Station
						tx_length2 	= 2
						WriteEnable2	= TRUE								;Set write enable
					ELSE
						tx_frame2[0] = $15 									;NAK
						tx_frame2[1] = rdata2[0] 							;PLC Station
						tx_length2 	 = 2
						WriteEnable2 = TRUE									;Set write enable
					ENDIF
				ENDIF

			ELSE

				tx_frame2[0] = $15 										;NAK
				tx_frame2[1] = rdata2[0] 								;PLC Station
				tx_length2 	 = 2
				WriteEnable2 = TRUE										;Set write enable

			ENDIF

			IF WriteEnable2 THEN
				TCPsend_2.enable = 1
    			TCPsend_2.cident = TCPserv_2.cident
    			TCPsend_2.buffer = ADR(tx_frame2[0])
    			TCPsend_2.buflng = tx_length2 ;SIZEOF(tx_frame)
    			TCPsend_2 FUB TCPsend()
	    	ENDIF

	    ENDIF

	ELSE
		TCPsend_2 FUB TCPsend()
	ENDIF

    IF (((TCPsend_2.status <> 0) AND (TCPsend_2.status <> 65535)) OR NoData2) THEN
    	NoData2  = FALSE
    	NEWSTEP2 = 4
    ENDIF

ENDIF
TON_10ms(((STEP2 = 3) AND (RXLength2 = 0)),500,NoData2,NoData2ET)

;Close the connection - if closed then go-to listen else go-to wait for close
IF STEP2 = 4 THEN
	TCPclose_2.enable = 1
	TCPclose_2.cident = TCPserv_2.cident
	TCPclose_2 FUB TCPclose()
	NEWSTEP2 = 5
ENDIF

;Closing - wait until connection closed
IF STEP2 = 5 THEN
	IF TCPclose_2.status <> 0 THEN
		TCPclose_2 FUB TCPclose()
	ELSE IF TCPclose_2.status = 0 THEN
		TCPsend_2.status = 0
		NEWSTEP2 = 1
	ENDIF
ENDIF

IF STEP2 = 6 THEN
	;Warm / Cold Start Required
ENDIF

;Clear Reset Connection from Init Sub
ResetConnection = FALSE
END_PROGRAM
```

### Program Logical/Sequences/10ms/zzIO (IEC) - * PLC Inputs and Outputs to Graphics

#### zzio.ab
```automation-basic
PROGRAM _CYCLIC
(* cyclic program *)

;Transmit I/O to PC Graphics

;-----------------------------------------------------------------------------------------
;Version 1.00 19/12/2005 D.J. First Issue
;Version 2.00 13/11/2006 D.J. All I/O Sent to Graphics
;Version 3.00 02/05/2007 D.J. Do more than 1 card per scan
;Version 4.00 20/11/2009 D.J. Changed from 16 I/O to 8 I/O Per Card (2 cards per 16-bit D)
;-----------------------------------------------------------------------------------------

LOOP n = 1 TO 5 DO ;Do 5 * 2 cards per scan

	CurrentCard 	= CurrentCard + 1
	DataRegister 	= DataRegister + 1

	IF (CurrentCard > Std.MaxIO) OR (DataRegister > 199) THEN
		CurrentCard = 0
		DataRegister = 0
	ENDIF

	InputCard.Input[0] 	= X[CurrentCard].X01
	InputCard.Input[1] 	= X[CurrentCard].X02
	InputCard.Input[2] 	= X[CurrentCard].X03
	InputCard.Input[3] 	= X[CurrentCard].X04
	InputCard.Input[4] 	= X[CurrentCard].X05
	InputCard.Input[5] 	= X[CurrentCard].X06
	InputCard.Input[6] 	= X[CurrentCard].X07
	InputCard.Input[7] 	= X[CurrentCard].X08
	InputCard.Input[8] 	= X[CurrentCard].X09
	InputCard.Input[9] 	= X[CurrentCard].X10
	InputCard.Input[10] = X[CurrentCard].X11
	InputCard.Input[11] = X[CurrentCard].X12
	InputCard.Input[12] = X[CurrentCard].X13
	InputCard.Input[13] = X[CurrentCard].X14
	InputCard.Input[14] = X[CurrentCard].X15
	InputCard.Input[15] = X[CurrentCard].X16
	InputCard FUB BIT_ENCODE()

	D[400 + DataRegister] 	= InputCard.Output

	OutputCard.Input[0] 	= Y[CurrentCard].Y01
	OutputCard.Input[1] 	= Y[CurrentCard].Y02
	OutputCard.Input[2] 	= Y[CurrentCard].Y03
	OutputCard.Input[3] 	= Y[CurrentCard].Y04
	OutputCard.Input[4] 	= Y[CurrentCard].Y05
	OutputCard.Input[5] 	= Y[CurrentCard].Y06
	OutputCard.Input[6] 	= Y[CurrentCard].Y07
	OutputCard.Input[7] 	= Y[CurrentCard].Y08
	OutputCard.Input[8] 	= Y[CurrentCard].Y09
	OutputCard.Input[9] 	= Y[CurrentCard].Y10
	OutputCard.Input[10] 	= Y[CurrentCard].Y11
	OutputCard.Input[11] 	= Y[CurrentCard].Y12
	OutputCard.Input[12] 	= Y[CurrentCard].Y13
	OutputCard.Input[13] 	= Y[CurrentCard].Y14
	OutputCard.Input[14] 	= Y[CurrentCard].Y15
	OutputCard.Input[15] 	= Y[CurrentCard].Y16
	OutputCard FUB BIT_ENCODE()

	D[600 + DataRegister] 	= OutputCard.Output

ENDLOOP
END_PROGRAM
```

### Program Logical/Sequences/10ms/zzOk (IEC) - * PLC Status to Graphics

#### zzok.ab
```automation-basic
PROGRAM _CYCLIC
(* cyclic program *)

;Transmit I/O Status to PC Graphics up-to 400 I/O Modules

;----------------------------------------
;Version 1.00 10/12/2007 D.J. First Issue
;----------------------------------------

Module = Module + 1

IF (Module > 3 ) THEN
	Module = 0
ENDIF

n = (Module * 16)

ModuleEncode.Input[0] 	= OK[n + 1]
ModuleEncode.Input[1] 	= OK[n + 2]
ModuleEncode.Input[2] 	= OK[n + 3]
ModuleEncode.Input[3] 	= OK[n + 4]
ModuleEncode.Input[4] 	= OK[n + 5]
ModuleEncode.Input[5] 	= OK[n + 6]
ModuleEncode.Input[6] 	= OK[n + 7]
ModuleEncode.Input[7] 	= OK[n + 8]
ModuleEncode.Input[8] 	= OK[n + 9]
ModuleEncode.Input[9] 	= OK[n + 10]
ModuleEncode.Input[10] 	= OK[n + 11]
ModuleEncode.Input[11] 	= OK[n + 12]
ModuleEncode.Input[12] 	= OK[n + 13]
ModuleEncode.Input[13] 	= OK[n + 14]
ModuleEncode.Input[14] 	= OK[n + 15]
ModuleEncode.Input[15] 	= OK[n + 16]
ModuleEncode FUB BIT_ENCODE()

D[320 + Module] 	= ModuleEncode.Output

StnModule = StnModule + 1

IF (StnModule > 3) THEN
	StnModule = 0
ENDIF

n = (StnModule * 16)

StnModuleEncode.Input[0] 	= StnOK[n + 1]
StnModuleEncode.Input[1] 	= StnOK[n + 2]
StnModuleEncode.Input[2] 	= StnOK[n + 3]
StnModuleEncode.Input[3] 	= StnOK[n + 4]
StnModuleEncode.Input[4] 	= StnOK[n + 5]
StnModuleEncode.Input[5] 	= StnOK[n + 6]
StnModuleEncode.Input[6] 	= StnOK[n + 7]
StnModuleEncode.Input[7] 	= StnOK[n + 8]
StnModuleEncode.Input[8] 	= StnOK[n + 9]
StnModuleEncode.Input[9] 	= StnOK[n + 10]
StnModuleEncode.Input[10] 	= StnOK[n + 11]
StnModuleEncode.Input[11] 	= StnOK[n + 12]
StnModuleEncode.Input[12] 	= StnOK[n + 13]
StnModuleEncode.Input[13] 	= StnOK[n + 14]
StnModuleEncode.Input[14] 	= StnOK[n + 15]
StnModuleEncode.Input[15] 	= StnOK[n + 16]
StnModuleEncode FUB BIT_ENCODE()

D[350 + StnModule] 	= StnModuleEncode.Output
END_PROGRAM
```

### Program Logical/Sequences/10ms/zzUld_4a (IEC, version 4.20.0)

#### zzuld_4.ab
```automation-basic
;Unloading Programs 4 - Search and give Destination (Using Bag)

	;-----------------------------------------------------------
	;Version 1.00 03/12/2005 D.J. First Issue
	;Version 2.00 30/08/2007 D.J. BagRemaining changed to INT
	;Version 3.00 25/06/2009 D.J. Use .Prg Instead of .Cat
	;Version 4.00 09/11/2009 D.J. Allow multiple destination
	;Version 4.10 08/06/2011 D.J. Addes Start/Stop for each line
	;-----------------------------------------------------------

PROGRAM _INIT

	;Constants
	;---------

	UnloadingMaxDepth 	= 7 ;Set with Batch Size and Scan Time in mind 8 = Standard

	StartDischarger 	= 3
	EndDischarger   	= 4 ;Allowed for 3rd future discharger so recirc takes dest 24

;	Line15Bags[1]			= 231
;	Line15Bags[2]			= 259
;	Line15Bags[3]			= 261
;	Line15Bags[4]			= 243
;	Line15Bags[5]			= 244
;	Line15Bags[6]			= 245
;	Line15Bags[7]			= 246

	StartLineSearch 	= 30
	EndLineSearch 		= 31;Include Lines A-C

	SkipLineStart		= 0
	SkipLineEnd			= 0

	RegOffset[1]    	= 1000
	RegOffset[2]    	= 1200
	RegOffset[3]    	= 1400
	RegOffset[4]    	= 1600
	RegOffset[5]    	= 1800
	RegOffset[6]    	= 2000
	RegOffset[7]    	= 2200
	RegOffset[8]    	= 2400

	;Enter Line Number for Discharger buffers - Recirc is after last Discharger
	;Destination Code bag will be allocated
	;BufferLineNum[1]	= 21
	;BufferLineNum[2]	= 22
	BufferLineNum[3]	= 23
	BufferLineNum[4]	= 24
	BufferLineNum[5]	= 0
	BufferLineNum[6]	= 0
	BufferLineNum[7]	= 0
	BufferLineNum[8]	= 0

	RecircDest			= 30

	PriorityLine		= 30		;Always Search this line first then use the Uld[n].DischargerStartLine Set to 0 if not required

	StartStopOffset		= 200	;Offset for D register for each lines Start / Stop ie D201 to D2xx - Set to Zero if no Start / Stops

END_PROGRAM

PROGRAM _CYCLIC

	pairingloopBIT = 0
	LOOP n=1 TO UnloadingMaxDepth DO
		IF (Bag[Line15Bags[n]].Dst = RecircDest) THEN
			INC pairingloopBIT //Offset is calculated as BIT for bags 1 to 4 is irrelevent
		ENDIF
	ENDLOOP

	;Spare Step
	IF (UldStep = 0) THEN
		UldStep = 1
	ENDIF

	;UldStep 1	- Check no bags in Storage are allocated with a destination
	IF (UldStep = 1) THEN

		;Set ScanCount as alternating Value 25 is about 5 seconds
		IF (ScanCount = 1) THEN
			Discharger 	= (Discharger + 1)
			ScanCount 	= 0
		ENDIF

		ScanCount = (ScanCount + 1)

		IF ((Discharger > EndDischarger) OR (Discharger < StartDischarger))  THEN
			Discharger 	= StartDischarger
		ENDIF

		;Set discharger number in TestDischarger if required
		IF (TestDischarger > 0) THEN
			Discharger = TestDischarger
		ENDIF

		;Read Program Variables
		n = RegOffset[Discharger]

		ProgramStep 			= D[1 + n]
		ProgQtyComplete			= D[2 + n]
		AutoRecirculation 		= (D[1003] = 1)		;Use if Re-cirulation or Offgoing Batching Loop
		RecirculationMaxDepth 	= D[1004]

		ManualLine       		= D[7 + n]
		ManualBags       		= D[8 + n]
		StepsSearched			= D[9 + n]
		SkipIncompleteStep 		= (D[10 + n] = 1)
		AutoRepeat				= (D[11 + n] = 1)
		MixPrograms 			= (D[12 + n] = 1)	;Batch must be same Program?
		MixCustomers 			= (D[13 + n] = 1) 	;Batch must be same Customer?
		NoBagAvailable			= (D[14 + n] = 1)	;Alarm 'No Bag Available'
		ProgramFinished			= (D[15 + n] = 1)	;Alarm 'Finished Program'
		ManualLineRecirc 		= D[1016]
		ManualBagsRecirc 		= D[1017]
		ProgramRunning			= (D[19 + n] = 1)	;Run from TrackView
		ExpressLine 			= D[20 + n]
		CustomerMode			= D[21 + n]			;Customer Mode 0 = Normal Manual, 1 = Reset Pointer on every step, 2 = Check all steps before changing
		ProgramReset			= (D[22 + n] = 1)	;Customer FIFO Reset

		DischargerReady			= Uld[Discharger].SDCReady

		DischargerSpaces = 5;Line[BufferLineNum[Discharger]].SpaceBIT
		;Calculate RecircSpaces
		RecircSpaces  		=  Line[RecircDest].Space - DestCountSystem[RecircDest] + pairingloopBIT
		IF (RecircSpaces < 0) THEN ; Keep value positive
			RecircSpaces = 0
		ENDIF
		BagsWithDest 			= Std.BagsWithDestinations2

		IF ((BagsWithDest = 0) AND (Discharger > 0)) THEN
			UldStep = 2
		ELSE
			;Allow program to skip blank steps when Bags Have Destinations
			UnusedStep		= (D[40 + n + ProgramStep] = 0) ;Bags = 0
			IF UnusedStep THEN
				UldStep = 15
			ENDIF
		ENDIF

		;If program is new then Clear Search Values
		IF ProgramReset THEN
			Uld[Discharger].FIFOCustomer 		= 0	;Clear Current Customer - FIFO Will allocate next
			Uld[Discharger].LastCustQtyComplete = 0	;Clear Last Quantity
			StepsSearched 						= 0	;Clear Steps Searched / Failed
			D[22 + n]	 						= 0 ;Clear Program Reset
			UldStep 							= 0	;Keep Unloading Step at 0 to allow Customer FIFO to allocate next Customer
		ENDIF

	ENDIF

	;UldStep 2	- Check for a Manual Re-circulation regardless of Discharger
	;			- Note will stop all unloading progrms if not ready
	IF (UldStep = 2) THEN
		IF ((ManualLineRecirc >= StartLineSearch) AND (ManualLineRecirc <= EndLineSearch) AND (ManualBagsRecirc > 0)) THEN
			IF Uld[EndDischarger + 1].SDCReady THEN
				UldStep = 21
			ELSE
				UldStep = 0
			ENDIF
		ELSE
			UldStep = 3
		ENDIF
	ENDIF

	;UldStep 3	- Check Discharger is Ready
	IF (UldStep = 3) THEN
		IF (DischargerReady AND ProgramRunning) THEN; AND (DischargerSpaces > 0)) THEN
			UldStep = 4
		ELSE
			;If not ready then clear steps searched
			UldStep = 0
		ENDIF
	ENDIF

	;UldStep 4	- Check for a Manual Bags
	IF (UldStep = 4) THEN
		IF ((ManualLine >= StartLineSearch) AND (ManualLine <= EndLineSearch) AND (ManualBags > 0)) THEN
			UldStep = 22
		ELSE
			UldStep = 5
		ENDIF
	ENDIF

	;STEP 5	- Check Express Line
	IF (UldStep = 5) THEN
		IF (ExpressLine > 0) THEN
			ExpressBag  = Line[ExpressLine].FirstBag
		ENDIF
		;IF ((Bag[ExpressBag].Cat > 0) AND (ExpressLine > 0) AND (Line[BufferLineNum[Discharger]].SpaceBIT > 0)) THEN
		IF ((Bag[ExpressBag].Cat > 0) AND (ExpressLine > 0) AND (Line[BufferLineNum[Discharger]].SpaceBIT > 0) AND (D[StartStopOffset + 7600 + ExpressLine] > 0)) THEN
			UldStep = 23
		ELSE
			UldStep = 6
		ENDIF
	ENDIF

	;UldStep 6	- Check Program step
	IF (UldStep = 6) THEN

		;Check if UldStep Valid
		IF (ProgramStep < 1) OR (ProgramStep > 20) THEN
			ProgramStep = 1 					;Set to UldStep 1
			ProgQtyComplete = 0 				;Clear Qty Completed
			IF (CustomerMode = 1) THEN
				Uld[Discharger].FIFOCustomer = 0
			ENDIF
		ENDIF

		UldStep = 7

	ENDIF

	;UldStep 7 - Check for remaining bags on the current Step
	IF (UldStep = 7) THEN

		BatchSize 		= D[80 + n + ProgramStep]
		Quantity 		= D[40 + n + ProgramStep] ;* BatchSize ;Take bags * BatchSize
		BagsRemaining 	= INT(Quantity - ProgQtyComplete)

		IF ((BagsRemaining > 0) AND (BagsRemaining >= INT(BatchSize))) THEN
			UldStep = 8
		ELSE
			UldStep = 15 ;Step Not Complete Or No Qty
		ENDIF

	ENDIF

	;UldStep 8 - Check the 'Batch' Will fit onto the Buffer
	IF (UldStep = 8) THEN

		BatchSize 		= D[80 + n + ProgramStep]

		IF (DischargerSpaces >= BatchSize) THEN
			UldStep = 9
		ELSE
			UldStep = 0
		ENDIF

	ENDIF

	;UldStep 9 - Set Search Values
	IF (UldStep = 9) THEN

		IF (PriorityLine = 0) THEN
			StartLine = (Uld[Discharger].DischargerStartLine + 1)
			IF ((StartLine < StartLineSearch) OR (StartLine > EndLineSearch)) THEN
				StartLine = StartLineSearch
			ENDIF
		ELSE
			StartLine = PriorityLine
		ENDIF

		SearchLine   = D[60 + n + ProgramStep]
		BatchSize    = D[80 + n + ProgramStep]

		SearchPrg[1] = D[100 + n + ProgramStep]
		SearchPrg[2] = D[120 + n + ProgramStep]
		SearchPrg[3] = D[140 + n + ProgramStep]

		IF (CustomerMode = 0) THEN
			SearchCus[1] = D32[20 + Discharger]					;Manually Selected Customer
		ELSE
			SearchCus[1] = Uld[Discharger].FIFOCustomer ;Automatic FIFO Customer Selection
		ENDIF

		SearchSpaces = 0 ;Search Always starts with no spaces on the recirc

		UldStep = 10

	ENDIF

	;UldStep 10 - Search for Bag(s) could be modified to run over several scans to reduce its load on the PLC
	;			  To find the best pos using set RecircSpaces low increasing to max.
	IF (UldStep = 10) THEN

		LOOP FindBest = 1 TO 3 DO

			;Clear the Search Array and Set Depth Allowed 1 for upto 49 storage lines
			FoundLine = 0
			memset(ADR(FoundBag[0]),0,10)
			memset(ADR(LineDepthAllowed[0]),1,50)

			RecircSpacesRemain = SearchSpaces

			;Can the 1st, 2nd or 3rd Program be mixed with each other? 'Mix Programs'
			IF (FindBest = 1) THEN
				MatchPrg1 = TRUE
				MatchPrg2 = FALSE
				MatchPrg3 = FALSE
			ELSE IF (FindBest = 2) THEN
				MatchPrg1 = MixPrograms
				MatchPrg2 = TRUE
				MatchPrg3 = FALSE
			ELSE
				MatchPrg1 = MixPrograms
				MatchPrg2 = MixPrograms
				MatchPrg3 = TRUE
			ENDIF

			;Loop around all the storage lins row by row.
			LOOP CurrentDepth = 1 TO UnloadingMaxDepth DO ;Always search to max depth to check scan time

				;CurrentLine = StartLine

				LOOP LinesSearched = StartLineSearch TO EndLineSearch DO ;Loop around each line
				 	CurrentLine = LinesSearched
					;CurrentLine = LongestTime[LinesSearched]
					CurrentBag = (Line[CurrentLine].FirstBag + (CurrentDepth - 1))
					//Special - Line 15 is pairing loop line bags are not in order. Declared at top
					IF LinesSearched = 15 THEN
						;CurrentBag = Line15Bags[CurrentDepth]
					ENDIF

					;Search / Add
					;------------
					;For Unloading by line - If there is a bag on the line and the 1st Program = 0 then check Customer valid
					;eg if the 1st Prg and 1st Cus are set to 0 then this would set "CatCusValid" to TRUE but the line must also match
					;Unloading by Customer only cannot be done.

					CatValid = (Bag[CurrentBag].Cat > 0)
					CusValid = FALSE
					PrgValid = FALSE
					DstValid = FALSE

					;Check the Destination is valid (allow dischargers to take recirc bags)
					IF ((Bag[CurrentBag].Dst = 0) OR (Bag[CurrentBag].Dst = RecircDest)) THEN
						DstValid = TRUE
					ENDIF

					;Check the Customer is valid
					IF (Bag[CurrentBag].Cus = SearchCus[1]) THEN
						CusValid = TRUE
					ELSE IF ((SearchCus[1] = 0) AND (CustomerMode = 0)) THEN ;Only Valid If Manual Customer Selection
						CusValid = TRUE
					ENDIF

					;Check the Category is valid
					IF (MatchPrg1 AND (Bag[CurrentBag].Prg = SearchPrg[1]) AND (SearchPrg[1] > 0)) THEN
						PrgValid = TRUE
					ENDIF
					IF (MatchPrg2 AND (Bag[CurrentBag].Prg = SearchPrg[2]) AND (SearchPrg[2] > 0)) THEN
						PrgValid = TRUE
					ENDIF
					IF (MatchPrg3 AND (Bag[CurrentBag].Prg = SearchPrg[3]) AND (SearchPrg[3] > 0)) THEN
						PrgValid = TRUE
					ENDIF
					;If Unloading by line and no Category is set then Set Valid
					IF ((Bag[CurrentBag].Cat > 0) AND (SearchPrg[1] = 0) AND (SearchLine > 0)) THEN
						PrgValid = TRUE
					ENDIF

					BagValid = (CurrentBag >= Line[CurrentLine].FirstBag) AND (CurrentBag <= Line[CurrentLine].LastBag)
					IF CurrentLine = 15 THEN
						BagValid = TRUE
					ENDIF

					LineValid 	= ((SearchLine = CurrentLine) OR (SearchLine = 0))
					LineValid2 	= ((CurrentLine < SkipLineStart) OR (CurrentLine > SkipLineEnd))
					IF (StartStopOffset < 100) THEN
						LineValid3	= ((StartStopOffset = 0) OR (D[StartStopOffset + CurrentLine] > 0))
					ELSE
						LineValid3	= (D[StartStopOffset + 7600 + CurrentLine] > 0) ;Start / Stop 100 -299 D7700 to D7899
					ENDIF

					DepthValid	= ((LineDepthAllowed[CurrentLine] + RecircSpacesRemain) >= CurrentDepth)
					DepthValid2	= ((CurrentDepth <= RecirculationMaxDepth) OR NOT AutoRecirculation)

;					IF CurrentLine = 15 THEN
;						DepthValid = Line[RecircDest].Space > 0
;						DepthValid2 = (CurrentDepth <= UnloadingMaxDepth)
;					ENDIF

					IF (BagValid AND DstValid AND CatValid AND PrgValid AND CusValid AND LineValid AND LineValid2 AND LineValid3 AND DepthValid AND DepthValid2) THEN

						IF (FoundBag[0] < BatchSize)  THEN
							FoundBag[0] = FoundBag[0] + 1
							x 			= FoundBag[0]
							FoundBag[x] = CurrentBag
							FoundLine	= CurrentLine

							;If bags need to go to recirc then dec
							IF (LineDepthAllowed[CurrentLine] < USINT(CurrentDepth)) THEN
								SpacesUsed 			= USINT(CurrentDepth) - LineDepthAllowed[CurrentLine]
								RecircSpacesRemain 	= (RecircSpacesRemain - SpacesUsed)
							ENDIF

							LineDepthAllowed[CurrentLine] = USINT(CurrentDepth + 1)

						ENDIF

					ENDIF

					;-------------
					;End of Search
					;-------------

					;If searching using priority line then start from the Discharger Start Line
					IF CurrentLine = PriorityLine THEN
						CurrentLine = (Uld[Discharger].DischargerStartLine)
					ENDIF

					;Set Next Line
					CurrentLine = (CurrentLine + 1)
					IF CurrentLine > EndLineSearch THEN
						CurrentLine = StartLineSearch
					ENDIF

					;If the new line = priority line then skip as its already been searched
					IF CurrentLine = PriorityLine THEN
						CurrentLine = (CurrentLine + 1)
						IF CurrentLine > EndLineSearch THEN
							CurrentLine = StartLineSearch
						ENDIF
					ENDIF

				ENDLOOP

			ENDLOOP

			EXITIF FoundBag[0] = BatchSize

		ENDLOOP				;Find Best

		;Check if the bags were found
		IF FoundBag[0] = BatchSize THEN
			UldStep = 14 	;Action Results
		ELSE IF (AutoRecirculation AND (RecircSpaces > SearchSpaces) AND (RecircSpaces > 0)) THEN
			;If recirculation - to find the best possible result inc the search spaces each scan
			;until total spaces searched
			SearchSpaces = (SearchSpaces + 1)
			UldStep = 10	;Try with more recirculation space
		ELSE
			UldStep = 15	;Search Failed
		ENDIF

	ENDIF

	;UldStep 14 - Search Valid give bags destinations, inc qty taken by batchsize
	IF (UldStep = 14) THEN

		LOOP Dest = 1 TO BatchSize DO
			Bag[FoundBag[Dest]].Dst = USINT(BufferLineNum[Discharger])
		ENDLOOP
		ProgQtyComplete = ProgQtyComplete + BatchSize	;Inc Qty Completed
		StepsSearched = 0 								;Clear the search failed UldStep counter
		NoBagAvailable = FALSE 							;No Bags Alarm (OFF)
		LastDischarger = Discharger

		IF AutoRecirculation THEN
			UldStep = 24		;Set Any Bags for Auto-Reirculation
		ELSE
			UldStep = 0
		ENDIF

		;Mode 2 Needs to keep the Qty completed for the next customer
		Uld[Discharger].LastCustQtyComplete = ProgQtyComplete

	ENDIF

	;UldStep 15 - Search Failed
	IF (UldStep = 15) THEN

		BatchSize 		= D[80 + n + ProgramStep]
		;Quantity 		= D[40 + n + ProgramStep] * BatchSize ;Take bags * BatchSize
		Quantity		= (D[40 + n + ProgramStep])
		BagsRemaining 	= INT(Quantity - ProgQtyComplete)
		UnusedStep		= (D[40 + n + ProgramStep] = 0) ;Bags = 0

		;Inc Steps searched counter
		IF (StepsSearched < 21) THEN
			StepsSearched = (StepsSearched + 1)
		ENDIF

		IF (CustomerMode = 0) THEN
			IF (BagsRemaining <= 0) THEN
				UldStep = 16			;Try Next Step
			ELSE IF (SkipIncompleteStep OR UnusedStep) THEN
				UldStep = 16			;Try Next Step
			ELSE
				NoBagAvailable = TRUE 	;Set Alarm and Wait for Operator to change Program or More Bags
				UldStep = 0
			ENDIF
		ENDIF

		IF (CustomerMode = 1) THEN
			IF (BagsRemaining <= 0) THEN
				UldStep = 16			;Try Next Step
			ELSE IF (NOT UnusedStep) THEN
				IF (Uld[Discharger].FIFONextCustomer > 0) THEN
					;Mode 1 Search again with the Next Customer Without Changing Step
					Uld[Discharger].FIFOCustomer = Uld[Discharger].FIFONextCustomer
					UldStep = 0
				ELSE
					;Last customer was not found reset FIFO position to 1 and keep searching
					Uld[Discharger].FIFOCustomer = 0 ;Reset the First Customer
					NoBagAvailable = TRUE
					UldStep = 0
				ENDIF
			ELSE IF (SkipIncompleteStep OR UnusedStep) THEN
				UldStep = 16			;Try Next Step
			ELSE
				NoBagAvailable = TRUE	;Set Alarm and Wait for Operator to change Program or More Bags
				UldStep = 0
			ENDIf
		ENDIF

		IF (CustomerMode = 2) THEN
			IF (BagsRemaining <= 0) THEN
				UldStep = 16			;Try Next Step
			ELSE IF (StepsSearched = 21) THEN
				IF (Uld[Discharger].FIFONextCustomer > 0) THEN
					;Mode 2 Customer Change Only After 21 Steps Searched
					Uld[Discharger].FIFOCustomer = Uld[Discharger].FIFONextCustomer
					ProgQtyComplete = Uld[Discharger].LastCustQtyComplete
					StepsSearched = 0 ;FREI Use -1 to go to next step
					UldStep = 0
				ELSE
					;Last customer was not found reset FIFO position to 1 and keep searching
					Uld[Discharger].FIFOCustomer = 0 ;Reset the First Customer
					NoBagAvailable = TRUE
					StepsSearched = 0
					UldStep = 0
				ENDIF
			ELSE IF (SkipIncompleteStep OR UnusedStep) THEN
				UldStep = 16			;Try Next Step
			ELSE
				NoBagAvailable = TRUE	;Set Alarm and Wait for Operator to change Program or More Bags
				UldStep = 0
			ENDIF
		ENDIF

	ENDIF

	;Skip Program Step or Set to 1
	IF (UldStep = 16) THEN
		IF (ProgramStep = 20) THEN
			IF AutoRepeat THEN
				ProgramStep = 1
				IF (CustomerMode = 1) THEN
					Uld[Discharger].FIFOCustomer = 0 ;Start Search With First Customer
				ENDIF
			ELSE
				ProgramFinished = TRUE
			ENDIF
		ELSE
			ProgramStep = ProgramStep + 1
			IF (CustomerMode = 1) THEN
				Uld[Discharger].FIFOCustomer = 0 ;Start Search With First Customer
			ENDIF
		ENDIF
		ProgQtyComplete = 0
		UldStep = 0
	ENDIF

	;UldStep 21 -	Manual Bags Recirc
	IF (UldStep = 21) THEN

		LOOP RecircBag = 0 TO (ManualBagsRecirc - 1) DO

			CurrentBag = (Line[ManualLineRecirc].FirstBag + RecircBag)

			IF Bag[CurrentBag].Cat > 0 THEN
				Bag[CurrentBag].Dst = USINT(RecircDest)	;Set Destination
				;ManualBagsRecirc    = (ManualBagsRecirc - 1)					;Dec manual bags by 1
			ENDIF
		ENDLOOP
		ManualBagsRecirc = 0
		UldStep = 0

	ENDIF

	;UldStep 22 - Manual Bags to Discharger
	IF (UldStep = 22) THEN

		CurrentBag = Line[ManualLine].FirstBag

		IF Bag[CurrentBag].Cat > 0 THEN
			Bag[CurrentBag].Dst = USINT(BufferLineNum[Discharger])
			ManualBags 			= (ManualBags - 1)				;Dec manual bags by 1
		ENDIF

		UldStep = 0

	ENDIF

	;UldStep 23 - Express Line
	IF (UldStep = 23) THEN

		Bag[ExpressBag].Dst = USINT(BufferLineNum[Discharger])

		UldStep = 0

	ENDIF

	;UldStep 24 - Set Bags to re-circulation line if they need to move out of the way of bags with destinations
	IF (UldStep = 24) THEN

		LOOP CurrentLine = StartLineSearch to EndLineSearch DO
			//Special - Line 15 is pairing loop line bags are not in order. Declared at top
			IF CurrentLine = 15 THEN
				LOOP CurrentBag = UnloadingMaxDepth DOWNTO 1 DO
					IF (CurrentBag > 1) THEN
						IF (Bag[Line15Bags[CurrentBag]].Dst > 0) AND (Bag[Line15Bags[CurrentBag-1]].Dst = 0) THEN
							Bag[Line15Bags[CurrentBag-1]].Dst = USINT(RecircDest)
						ENDIF
					ENDIF
				ENDLOOP
			ELSE
				LOOP CurrentBag = Line[CurrentLine].LastBag DOWNTO Line[CurrentLine].FirstBag DO
					IF (CurrentBag > 0) THEN
						IF (Bag[CurrentBag].Dst > 0) AND (Bag[CurrentBag - 1].Dst = 0) AND (CurrentBag > Line[CurrentLine].FirstBag) THEN
							Bag[CurrentBag - 1].Dst = USINT(RecircDest)
						ENDIF
					ENDIF
				ENDLOOP
			ENDIF
		ENDLOOP

		UldStep = 0

	ENDIF

	;Outputs
	;-------

	D[1 + n] 		= ProgramStep
	D[2 + n]		= ProgQtyComplete
	D[8 + n] 		= ManualBags
	D[9 + n]		= StepsSearched

	;No bag available is displayed if 20 steps have been searched and program is running
	IF (NoBagAvailable AND ProgramRunning) THEN
		D[14 + n] = 1
		Alarm[Discharger + 200].On		= TRUE
		Alarm[Discharger + 200].Bag 	= 0
		Alarm[Discharger + 200].Name 	= almUldNoBag
		Alarm[Discharger + 200].Beacon	= FALSE
	ELSE
		D[14 + n]	= 0
	ENDIF

	;Program is only finished if on step 20 and Program Running
	IF (ProgramFinished AND ProgramRunning AND (ProgramStep = 20)) THEN
		D[15 + n]	= 1
		Alarm[Discharger + 200].On		= TRUE
		Alarm[Discharger + 200].Bag 	= 0
		Alarm[Discharger + 200].Name 	= almUldProgFinished
		Alarm[Discharger + 200].Beacon	= FALSE
	ELSE
		D[15 + n]	= 0
	ENDIF

	;If no unloading alarms then clear unloading alarm
	IF (D[14 + n] = 0) AND (D[15 + n] = 0) THEN
		Alarm[Discharger + 200].On		= FALSE
		Alarm[Discharger + 200].Bag 	= 0
		Alarm[Discharger + 200].Name 	= almNoAlarm
		Alarm[Discharger + 200].Beacon	= FALSE
	ENDIF

	D[1017]		= ManualBagsRecirc

	IF ProgramRunning THEN
		D[18 + n]	= 1
	ELSE
		D[18 + n]	= 0
	ENDIF

	D32[30 + Discharger] 	= Uld[Discharger].FIFOCustomer
	;D[187 + n] 		= Uld[Discharger].FIFONextCustomer

END_PROGRAM
```

### Program Logical/Sequences/10ms/zzUld_4 (IEC, version 4.20.0)

#### zzuld_4.var
```iecst
VAR
	AutoRecirculation : BOOL;
END_VAR
VAR RETAIN
	AutoRepeat : BOOL;
	BagsRemaining : INT;
	BatchSize : UINT;
	BufferLineNum : ARRAY[0..19] OF UINT;
	PrgValid : BOOL;
	CurrentBag : UINT;
	CurrentDepth : UINT;
	CurrentLine : UINT;
	CustomerMode : UINT;
	CusValid : BOOL;
	DepthValid : BOOL;
	DepthValid2 : BOOL;
	Dest : UINT;
	Discharger : UINT;
	DischargerReady : BOOL;
	DischargerSpaces : INT;
	EndDischarger : UINT;
	EndLineSearch : UINT;
	ExpressBag : UINT;
	ExpressLine : UINT;
	FindBest : UINT;
	FoundBag : ARRAY[0..4] OF UINT;
	FoundLine : UINT;
	LastDischarger : UINT;
	LineDepthAllowed : ARRAY[0..49] OF USINT;
	LinesSearched : UINT;
	LineValid : BOOL;
	ManualBags : UINT;
	ManualBagsRecirc : UINT;
	ManualLine : UINT;
	ManualLineRecirc : UINT;
	MatchPrg1 : BOOL;
	MatchPrg2 : BOOL;
	MatchPrg3 : BOOL;
	MixCustomers : BOOL;
	n : UINT;
	NoBagAvailable : BOOL;
	PLS : BOOL;
	PriorityLine : UINT;
	ProgQtyComplete : UINT;
	ProgramFinished : BOOL;
	ProgramReset : BOOL;
	ProgramRunning : BOOL;
	ProgramStep : UINT;
	Quantity : UINT;
	RecircDest : UINT;
	RecircSpaces : INT;
	RecircSpacesRemain : UINT;
	RecirculationMaxDepth : UINT;
	RegOffset : ARRAY[0..19] OF UINT;
	ScanCount : UINT;
	SearchPrg : ARRAY[0..3] OF UINT;
	SearchCus : ARRAY[0..3] OF UDINT;
	SearchLine : UINT;
	SearchSpaces : UINT;
	SkipIncompleteStep : BOOL;
	SpacesUsed : UINT;
	StartDischarger : UINT;
	StartLine : UINT;
	StartLineSearch : UINT;
	StepsSearched : UINT;
	TestDischarger : UINT;
	UldStep : UINT;
END_VAR
VAR
	UnloadingMaxDepth : UINT;
END_VAR
VAR RETAIN
	UnusedStep : BOOL;
	x : UINT;
	MixPrograms : BOOL;
END_VAR
VAR
	CatValid : BOOL;
	BagsWithDest : UINT;
	DstValid : BOOL;
	RecircLimit : INT;
	SkipLineStart : UINT;
	SkipLineEnd : UINT;
	LineValid2 : BOOL;
	BagValid : BOOL;
	DischLimit : UINT;
	StartStopOffset : UINT;
	LineValid3 : BOOL;
	TimTest : UINT;
	TestPLS : BOOL;
	RecircBag : UINT;
	kein : UINT;
	kev : BOOL;
	Line15Bags : ARRAY[0..8] OF UINT;
	pairingloopBIT : USINT;
END_VAR
```

#### zzuld_4.ab
```automation-basic
;Unloading Programs 4 - Search and give Destination (Using Bag)

	;-----------------------------------------------------------
	;Version 1.00 03/12/2005 D.J. First Issue
	;Version 2.00 30/08/2007 D.J. BagRemaining changed to INT
	;Version 3.00 25/06/2009 D.J. Use .Prg Instead of .Cat
	;Version 4.00 09/11/2009 D.J. Allow multiple destination
	;Version 4.10 08/06/2011 D.J. Addes Start/Stop for each line
	;-----------------------------------------------------------

PROGRAM _INIT

	;Constants
	;---------

	UnloadingMaxDepth 	= 7 ;Set with Batch Size and Scan Time in mind 8 = Standard

	StartDischarger 	= 1
	EndDischarger   	= 4 ;Allowed for 3rd future discharger so recirc takes dest 24

;	Line15Bags[1]			= 231
;	Line15Bags[2]			= 259
;	Line15Bags[3]			= 261
;	Line15Bags[4]			= 243
;	Line15Bags[5]			= 244
;	Line15Bags[6]			= 245
;	Line15Bags[7]			= 246

	StartLineSearch 	= 1
	EndLineSearch 		= 6 ;Include Lines A-C

	SkipLineStart		= 0
	SkipLineEnd			= 0

	RegOffset[1]    	= 1000
	RegOffset[2]    	= 1200
	RegOffset[3]    	= 1400
	RegOffset[4]    	= 1600
	RegOffset[5]    	= 1800
	RegOffset[6]    	= 2000
	RegOffset[7]    	= 2200
	RegOffset[8]    	= 2400

	;Enter Line Number for Discharger buffers - Recirc is after last Discharger
	;Destination Code bag will be allocated
	BufferLineNum[1]	= 11
	BufferLineNum[2]	= 12
	BufferLineNum[3]	= 13
	BufferLineNum[4]	= 0
	BufferLineNum[5]	= 0
	BufferLineNum[6]	= 0
	BufferLineNum[7]	= 0
	BufferLineNum[8]	= 0

	RecircDest			= 30

	PriorityLine		= 15		;Always Search this line first then use the Uld[n].DischargerStartLine Set to 0 if not required

	StartStopOffset		= 200	;Offset for D register for each lines Start / Stop ie D201 to D2xx - Set to Zero if no Start / Stops

END_PROGRAM

PROGRAM _CYCLIC

	pairingloopBIT = 0
	LOOP n=1 TO UnloadingMaxDepth DO
		IF (Bag[Line15Bags[n]].Dst = RecircDest) THEN
			INC pairingloopBIT //Offset is calculated as BIT for bags 1 to 4 is irrelevent
		ENDIF
	ENDLOOP

	;Spare Step
	IF (UldStep = 0) THEN
		UldStep = 1
	ENDIF

	;UldStep 1	- Check no bags in Storage are allocated with a destination
	IF (UldStep = 1) THEN

		;Set ScanCount as alternating Value 25 is about 5 seconds
		IF (ScanCount = 1) THEN
			Discharger 	= (Discharger + 1)
			ScanCount 	= 0
		ENDIF

		ScanCount = (ScanCount + 1)

		IF ((Discharger > EndDischarger) OR (Discharger < StartDischarger))  THEN
			Discharger 	= StartDischarger
		ENDIF

		;Set discharger number in TestDischarger if required
		IF (TestDischarger > 0) THEN
			Discharger = TestDischarger
		ENDIF

		;Read Program Variables
		n = RegOffset[Discharger]

		ProgramStep 			= D[1 + n]
		ProgQtyComplete			= D[2 + n]
		AutoRecirculation 		= (D[1003] = 1)		;Use if Re-cirulation or Offgoing Batching Loop
		RecirculationMaxDepth 	= D[1004]

		ManualLine       		= D[7 + n]
		ManualBags       		= D[8 + n]
		StepsSearched			= D[9 + n]
		SkipIncompleteStep 		= (D[10 + n] = 1)
		AutoRepeat				= (D[11 + n] = 1)
		MixPrograms 			= (D[12 + n] = 1)	;Batch must be same Program?
		MixCustomers 			= (D[13 + n] = 1) 	;Batch must be same Customer?
		NoBagAvailable			= (D[14 + n] = 1)	;Alarm 'No Bag Available'
		ProgramFinished			= (D[15 + n] = 1)	;Alarm 'Finished Program'
		ManualLineRecirc 		= D[1016]
		ManualBagsRecirc 		= D[1017]
		ProgramRunning			= (D[19 + n] = 1)	;Run from TrackView
		ExpressLine 			= D[20 + n]
		CustomerMode			= D[21 + n]			;Customer Mode 0 = Normal Manual, 1 = Reset Pointer on every step, 2 = Check all steps before changing
		ProgramReset			= (D[22 + n] = 1)	;Customer FIFO Reset

		DischargerReady			= Uld[Discharger].SDCReady

		DischargerSpaces = Line[BufferLineNum[Discharger]].SpaceBIT
		;Calculate RecircSpaces
		RecircSpaces  		=  Line[RecircDest].Space - DestCountSystem[RecircDest] + pairingloopBIT
		IF (RecircSpaces < 0) THEN ; Keep value positive
			RecircSpaces = 0
		ENDIF
		BagsWithDest 			= DestCountStorage[BufferLineNum[Discharger]]

		IF ((BagsWithDest = 0) AND (Discharger > 0)) THEN
			UldStep = 2
		ELSE
			;Allow program to skip blank steps when Bags Have Destinations
			UnusedStep		= (D[40 + n + ProgramStep] = 0) ;Bags = 0
			IF UnusedStep THEN
				UldStep = 15
			ENDIF
		ENDIF

		;If program is new then Clear Search Values
		IF ProgramReset THEN
			Uld[Discharger].FIFOCustomer 		= 0	;Clear Current Customer - FIFO Will allocate next
			Uld[Discharger].LastCustQtyComplete = 0	;Clear Last Quantity
			StepsSearched 						= 0	;Clear Steps Searched / Failed
			D[22 + n]	 						= 0 ;Clear Program Reset
			UldStep 							= 0	;Keep Unloading Step at 0 to allow Customer FIFO to allocate next Customer
		ENDIF

	ENDIF

	;UldStep 2	- Check for a Manual Re-circulation regardless of Discharger
	;			- Note will stop all unloading progrms if not ready
	IF (UldStep = 2) THEN
		IF ((ManualLineRecirc >= StartLineSearch) AND (ManualLineRecirc <= EndLineSearch) AND (ManualBagsRecirc > 0)) THEN
			IF Uld[EndDischarger + 1].SDCReady THEN
				UldStep = 21
			ELSE
				UldStep = 0
			ENDIF
		ELSE
			UldStep = 3
		ENDIF
	ENDIF

	;UldStep 3	- Check Discharger is Ready
	IF (UldStep = 3) THEN
		IF (DischargerReady AND ProgramRunning) THEN; AND (DischargerSpaces > 0)) THEN
			UldStep = 4
		ELSE
			;If not ready then clear steps searched
			UldStep = 0
		ENDIF
	ENDIF

	;UldStep 4	- Check for a Manual Bags
	IF (UldStep = 4) THEN
		IF ((ManualLine >= StartLineSearch) AND (ManualLine <= EndLineSearch) AND (ManualBags > 0)) THEN
			UldStep = 22
		ELSE
			UldStep = 5
		ENDIF
	ENDIF

	;STEP 5	- Check Express Line
	IF (UldStep = 5) THEN
		IF (ExpressLine > 0) THEN
			ExpressBag  = Line[ExpressLine].FirstBag
		ENDIF
		;IF ((Bag[ExpressBag].Cat > 0) AND (ExpressLine > 0) AND (Line[BufferLineNum[Discharger]].SpaceBIT > 0)) THEN
		IF ((Bag[ExpressBag].Cat > 0) AND (ExpressLine > 0) AND (Line[BufferLineNum[Discharger]].SpaceBIT > 0) AND (D[StartStopOffset + 7600 + ExpressLine] > 0)) THEN
			UldStep = 23
		ELSE
			UldStep = 6
		ENDIF
	ENDIF

	;UldStep 6	- Check Program step
	IF (UldStep = 6) THEN

		;Check if UldStep Valid
		IF (ProgramStep < 1) OR (ProgramStep > 20) THEN
			ProgramStep = 1 					;Set to UldStep 1
			ProgQtyComplete = 0 				;Clear Qty Completed
			IF (CustomerMode = 1) THEN
				Uld[Discharger].FIFOCustomer = 0
			ENDIF
		ENDIF

		UldStep = 7

	ENDIF

	;UldStep 7 - Check for remaining bags on the current Step
	IF (UldStep = 7) THEN

		BatchSize 		= D[80 + n + ProgramStep]
		Quantity 		= D[40 + n + ProgramStep] ;* BatchSize ;Take bags * BatchSize
		BagsRemaining 	= INT(Quantity - ProgQtyComplete)

		IF ((BagsRemaining > 0) AND (BagsRemaining >= INT(BatchSize))) THEN
			UldStep = 8
		ELSE
			UldStep = 15 ;Step Not Complete Or No Qty
		ENDIF

	ENDIF

	;UldStep 8 - Check the 'Batch' Will fit onto the Buffer
	IF (UldStep = 8) THEN

		BatchSize 		= D[80 + n + ProgramStep]

		IF (DischargerSpaces >= BatchSize) THEN
			UldStep = 9
		ELSE
			UldStep = 0
		ENDIF

	ENDIF

	;UldStep 9 - Set Search Values
	IF (UldStep = 9) THEN

		IF (PriorityLine = 0) THEN
			StartLine = (Uld[Discharger].DischargerStartLine + 1)
			IF ((StartLine < StartLineSearch) OR (StartLine > EndLineSearch)) THEN
				StartLine = StartLineSearch
			ENDIF
		ELSE
			StartLine = PriorityLine
		ENDIF

		SearchLine   = D[60 + n + ProgramStep]
		BatchSize    = D[80 + n + ProgramStep]

		SearchPrg[1] = D[100 + n + ProgramStep]
		SearchPrg[2] = D[120 + n + ProgramStep]
		SearchPrg[3] = D[140 + n + ProgramStep]

		IF (CustomerMode = 0) THEN
			SearchCus[1] = D32[20 + Discharger]					;Manually Selected Customer
		ELSE
			SearchCus[1] = Uld[Discharger].FIFOCustomer ;Automatic FIFO Customer Selection
		ENDIF

		SearchSpaces = 0 ;Search Always starts with no spaces on the recirc

		UldStep = 10

	ENDIF

	;UldStep 10 - Search for Bag(s) could be modified to run over several scans to reduce its load on the PLC
	;			  To find the best pos using set RecircSpaces low increasing to max.
	IF (UldStep = 10) THEN

		LOOP FindBest = 1 TO 3 DO

			;Clear the Search Array and Set Depth Allowed 1 for upto 49 storage lines
			FoundLine = 0
			memset(ADR(FoundBag[0]),0,10)
			memset(ADR(LineDepthAllowed[0]),1,50)

			RecircSpacesRemain = SearchSpaces

			;Can the 1st, 2nd or 3rd Program be mixed with each other? 'Mix Programs'
			IF (FindBest = 1) THEN
				MatchPrg1 = TRUE
				MatchPrg2 = FALSE
				MatchPrg3 = FALSE
			ELSE IF (FindBest = 2) THEN
				MatchPrg1 = MixPrograms
				MatchPrg2 = TRUE
				MatchPrg3 = FALSE
			ELSE
				MatchPrg1 = MixPrograms
				MatchPrg2 = MixPrograms
				MatchPrg3 = TRUE
			ENDIF

			;Loop around all the storage lins row by row.
			LOOP CurrentDepth = 1 TO UnloadingMaxDepth DO ;Always search to max depth to check scan time

				;CurrentLine = StartLine

				LOOP LinesSearched = StartLineSearch TO EndLineSearch DO ;Loop around each line
				 	CurrentLine = LinesSearched
					;CurrentLine = LongestTime[LinesSearched]
					CurrentBag = (Line[CurrentLine].FirstBag + (CurrentDepth - 1))
					//Special - Line 15 is pairing loop line bags are not in order. Declared at top
					IF LinesSearched = 15 THEN
						;CurrentBag = Line15Bags[CurrentDepth]
					ENDIF

					;Search / Add
					;------------
					;For Unloading by line - If there is a bag on the line and the 1st Program = 0 then check Customer valid
					;eg if the 1st Prg and 1st Cus are set to 0 then this would set "CatCusValid" to TRUE but the line must also match
					;Unloading by Customer only cannot be done.

					CatValid = (Bag[CurrentBag].Cat > 0)
					CusValid = FALSE
					PrgValid = FALSE
					DstValid = FALSE

					;Check the Destination is valid (allow dischargers to take recirc bags)
					IF ((Bag[CurrentBag].Dst = 0) OR (Bag[CurrentBag].Dst = RecircDest)) THEN
						DstValid = TRUE
					ENDIF

					;Check the Customer is valid
					IF (Bag[CurrentBag].Cus = SearchCus[1]) THEN
						CusValid = TRUE
					ELSE IF ((SearchCus[1] = 0) AND (CustomerMode = 0)) THEN ;Only Valid If Manual Customer Selection
						CusValid = TRUE
					ENDIF

					;Check the Category is valid
					IF (MatchPrg1 AND (Bag[CurrentBag].Prg = SearchPrg[1]) AND (SearchPrg[1] > 0)) THEN
						PrgValid = TRUE
					ENDIF
					IF (MatchPrg2 AND (Bag[CurrentBag].Prg = SearchPrg[2]) AND (SearchPrg[2] > 0)) THEN
						PrgValid = TRUE
					ENDIF
					IF (MatchPrg3 AND (Bag[CurrentBag].Prg = SearchPrg[3]) AND (SearchPrg[3] > 0)) THEN
						PrgValid = TRUE
					ENDIF
					;If Unloading by line and no Category is set then Set Valid
					IF ((Bag[CurrentBag].Cat > 0) AND (SearchPrg[1] = 0) AND (SearchLine > 0)) THEN
						PrgValid = TRUE
					ENDIF

					BagValid = (CurrentBag >= Line[CurrentLine].FirstBag) AND (CurrentBag <= Line[CurrentLine].LastBag)
					IF CurrentLine = 15 THEN
						BagValid = TRUE
					ENDIF

					LineValid 	= ((SearchLine = CurrentLine) OR (SearchLine = 0))
					LineValid2 	= ((CurrentLine < SkipLineStart) OR (CurrentLine > SkipLineEnd))
					IF (StartStopOffset < 100) THEN
						LineValid3	= ((StartStopOffset = 0) OR (D[StartStopOffset + CurrentLine] > 0))
					ELSE
						LineValid3	= (D[StartStopOffset + 7600 + CurrentLine] > 0) ;Start / Stop 100 -299 D7700 to D7899
					ENDIF

					DepthValid	= ((LineDepthAllowed[CurrentLine] + RecircSpacesRemain) >= CurrentDepth)
					DepthValid2	= ((CurrentDepth <= RecirculationMaxDepth) OR NOT AutoRecirculation)

;					IF CurrentLine = 15 THEN
;						DepthValid = Line[RecircDest].Space > 0
;						DepthValid2 = (CurrentDepth <= UnloadingMaxDepth)
;					ENDIF

					IF (BagValid AND DstValid AND CatValid AND PrgValid AND CusValid AND LineValid AND LineValid2 AND LineValid3 AND DepthValid AND DepthValid2) THEN

						IF (FoundBag[0] < BatchSize)  THEN
							FoundBag[0] = FoundBag[0] + 1
							x 			= FoundBag[0]
							FoundBag[x] = CurrentBag
							FoundLine	= CurrentLine

							;If bags need to go to recirc then dec
							IF (LineDepthAllowed[CurrentLine] < USINT(CurrentDepth)) THEN
								SpacesUsed 			= USINT(CurrentDepth) - LineDepthAllowed[CurrentLine]
								RecircSpacesRemain 	= (RecircSpacesRemain - SpacesUsed)
							ENDIF

							LineDepthAllowed[CurrentLine] = USINT(CurrentDepth + 1)

						ENDIF

					ENDIF

					;-------------
					;End of Search
					;-------------

					;If searching using priority line then start from the Discharger Start Line
					IF CurrentLine = PriorityLine THEN
						CurrentLine = (Uld[Discharger].DischargerStartLine)
					ENDIF

					;Set Next Line
					CurrentLine = (CurrentLine + 1)
					IF CurrentLine > EndLineSearch THEN
						CurrentLine = StartLineSearch
					ENDIF

					;If the new line = priority line then skip as its already been searched
					IF CurrentLine = PriorityLine THEN
						CurrentLine = (CurrentLine + 1)
						IF CurrentLine > EndLineSearch THEN
							CurrentLine = StartLineSearch
						ENDIF
					ENDIF

				ENDLOOP

			ENDLOOP

			EXITIF FoundBag[0] = BatchSize

		ENDLOOP				;Find Best

		;Check if the bags were found
		IF FoundBag[0] = BatchSize THEN
			UldStep = 14 	;Action Results
		ELSE IF (AutoRecirculation AND (RecircSpaces > SearchSpaces) AND (RecircSpaces > 0)) THEN
			;If recirculation - to find the best possible result inc the search spaces each scan
			;until total spaces searched
			SearchSpaces = (SearchSpaces + 1)
			UldStep = 10	;Try with more recirculation space
		ELSE
			UldStep = 15	;Search Failed
		ENDIF

	ENDIF

	;UldStep 14 - Search Valid give bags destinations, inc qty taken by batchsize
	IF (UldStep = 14) THEN

		LOOP Dest = 1 TO BatchSize DO
			Bag[FoundBag[Dest]].Dst = USINT(BufferLineNum[Discharger])
		ENDLOOP
		ProgQtyComplete = ProgQtyComplete + BatchSize	;Inc Qty Completed
		StepsSearched = 0 								;Clear the search failed UldStep counter
		NoBagAvailable = FALSE 							;No Bags Alarm (OFF)
		LastDischarger = Discharger

		IF AutoRecirculation THEN
			UldStep = 24		;Set Any Bags for Auto-Reirculation
		ELSE
			UldStep = 0
		ENDIF

		;Mode 2 Needs to keep the Qty completed for the next customer
		Uld[Discharger].LastCustQtyComplete = ProgQtyComplete

	ENDIF

	;UldStep 15 - Search Failed
	IF (UldStep = 15) THEN

		BatchSize 		= D[80 + n + ProgramStep]
		;Quantity 		= D[40 + n + ProgramStep] * BatchSize ;Take bags * BatchSize
		Quantity		= (D[40 + n + ProgramStep])
		BagsRemaining 	= INT(Quantity - ProgQtyComplete)
		UnusedStep		= (D[40 + n + ProgramStep] = 0) ;Bags = 0

		;Inc Steps searched counter
		IF (StepsSearched < 21) THEN
			StepsSearched = (StepsSearched + 1)
		ENDIF

		IF (CustomerMode = 0) THEN
			IF (BagsRemaining <= 0) THEN
				UldStep = 16			;Try Next Step
			ELSE IF (SkipIncompleteStep OR UnusedStep) THEN
				UldStep = 16			;Try Next Step
			ELSE
				NoBagAvailable = TRUE 	;Set Alarm and Wait for Operator to change Program or More Bags
				UldStep = 0
			ENDIF
		ENDIF

		IF (CustomerMode = 1) THEN
			IF (BagsRemaining <= 0) THEN
				UldStep = 16			;Try Next Step
			ELSE IF (NOT UnusedStep) THEN
				IF (Uld[Discharger].FIFONextCustomer > 0) THEN
					;Mode 1 Search again with the Next Customer Without Changing Step
					Uld[Discharger].FIFOCustomer = Uld[Discharger].FIFONextCustomer
					UldStep = 0
				ELSE
					;Last customer was not found reset FIFO position to 1 and keep searching
					Uld[Discharger].FIFOCustomer = 0 ;Reset the First Customer
					NoBagAvailable = TRUE
					UldStep = 0
				ENDIF
			ELSE IF (SkipIncompleteStep OR UnusedStep) THEN
				UldStep = 16			;Try Next Step
			ELSE
				NoBagAvailable = TRUE	;Set Alarm and Wait for Operator to change Program or More Bags
				UldStep = 0
			ENDIf
		ENDIF

		IF (CustomerMode = 2) THEN
			IF (BagsRemaining <= 0) THEN
				UldStep = 16			;Try Next Step
			ELSE IF (StepsSearched = 21) THEN
				IF (Uld[Discharger].FIFONextCustomer > 0) THEN
					;Mode 2 Customer Change Only After 21 Steps Searched
					Uld[Discharger].FIFOCustomer = Uld[Discharger].FIFONextCustomer
					ProgQtyComplete = Uld[Discharger].LastCustQtyComplete
					StepsSearched = 0 ;FREI Use -1 to go to next step
					UldStep = 0
				ELSE
					;Last customer was not found reset FIFO position to 1 and keep searching
					Uld[Discharger].FIFOCustomer = 0 ;Reset the First Customer
					NoBagAvailable = TRUE
					StepsSearched = 0
					UldStep = 0
				ENDIF
			ELSE IF (SkipIncompleteStep OR UnusedStep) THEN
				UldStep = 16			;Try Next Step
			ELSE
				NoBagAvailable = TRUE	;Set Alarm and Wait for Operator to change Program or More Bags
				UldStep = 0
			ENDIF
		ENDIF

	ENDIF

	;Skip Program Step or Set to 1
	IF (UldStep = 16) THEN
		IF (ProgramStep = 20) THEN
			IF AutoRepeat THEN
				ProgramStep = 1
				IF (CustomerMode = 1) THEN
					Uld[Discharger].FIFOCustomer = 0 ;Start Search With First Customer
				ENDIF
			ELSE
				ProgramFinished = TRUE
			ENDIF
		ELSE
			ProgramStep = ProgramStep + 1
			IF (CustomerMode = 1) THEN
				Uld[Discharger].FIFOCustomer = 0 ;Start Search With First Customer
			ENDIF
		ENDIF
		ProgQtyComplete = 0
		UldStep = 0
	ENDIF

	;UldStep 21 -	Manual Bags Recirc
	IF (UldStep = 21) THEN

		LOOP RecircBag = 0 TO (ManualBagsRecirc - 1) DO

			CurrentBag = (Line[ManualLineRecirc].FirstBag + RecircBag)

			IF Bag[CurrentBag].Cat > 0 THEN
				Bag[CurrentBag].Dst = USINT(RecircDest)	;Set Destination
				;ManualBagsRecirc    = (ManualBagsRecirc - 1)					;Dec manual bags by 1
			ENDIF
		ENDLOOP
		ManualBagsRecirc = 0
		UldStep = 0

	ENDIF

	;UldStep 22 - Manual Bags to Discharger
	IF (UldStep = 22) THEN

		CurrentBag = Line[ManualLine].FirstBag

		IF Bag[CurrentBag].Cat > 0 THEN
			Bag[CurrentBag].Dst = USINT(BufferLineNum[Discharger])
			ManualBags 			= (ManualBags - 1)				;Dec manual bags by 1
		ENDIF

		UldStep = 0

	ENDIF

	;UldStep 23 - Express Line
	IF (UldStep = 23) THEN

		Bag[ExpressBag].Dst = USINT(BufferLineNum[Discharger])

		UldStep = 0

	ENDIF

	;UldStep 24 - Set Bags to re-circulation line if they need to move out of the way of bags with destinations
	IF (UldStep = 24) THEN

		LOOP CurrentLine = StartLineSearch to EndLineSearch DO
			//Special - Line 15 is pairing loop line bags are not in order. Declared at top
			IF CurrentLine = 15 THEN
				LOOP CurrentBag = UnloadingMaxDepth DOWNTO 1 DO
					IF (CurrentBag > 1) THEN
						IF (Bag[Line15Bags[CurrentBag]].Dst > 0) AND (Bag[Line15Bags[CurrentBag-1]].Dst = 0) THEN
							Bag[Line15Bags[CurrentBag-1]].Dst = USINT(RecircDest)
						ENDIF
					ENDIF
				ENDLOOP
			ELSE
				LOOP CurrentBag = Line[CurrentLine].LastBag DOWNTO Line[CurrentLine].FirstBag DO
					IF (CurrentBag > 0) THEN
						IF (Bag[CurrentBag].Dst > 0) AND (Bag[CurrentBag - 1].Dst = 0) AND (CurrentBag > Line[CurrentLine].FirstBag) THEN
							Bag[CurrentBag - 1].Dst = USINT(RecircDest)
						ENDIF
					ENDIF
				ENDLOOP
			ENDIF
		ENDLOOP

		UldStep = 0

	ENDIF

	;Outputs
	;-------

	D[1 + n] 		= ProgramStep
	D[2 + n]		= ProgQtyComplete
	D[8 + n] 		= ManualBags
	D[9 + n]		= StepsSearched

	;No bag available is displayed if 20 steps have been searched and program is running
	IF (NoBagAvailable AND ProgramRunning) THEN
		D[14 + n] = 1
		Alarm[Discharger + 200].On		= TRUE
		Alarm[Discharger + 200].Bag 	= 0
		Alarm[Discharger + 200].Name 	= almUldNoBag
		Alarm[Discharger + 200].Beacon	= FALSE
	ELSE
		D[14 + n]	= 0
	ENDIF

	;Program is only finished if on step 20 and Program Running
	IF (ProgramFinished AND ProgramRunning AND (ProgramStep = 20)) THEN
		D[15 + n]	= 1
		Alarm[Discharger + 200].On		= TRUE
		Alarm[Discharger + 200].Bag 	= 0
		Alarm[Discharger + 200].Name 	= almUldProgFinished
		Alarm[Discharger + 200].Beacon	= FALSE
	ELSE
		D[15 + n]	= 0
	ENDIF

	;If no unloading alarms then clear unloading alarm
	IF (D[14 + n] = 0) AND (D[15 + n] = 0) THEN
		Alarm[Discharger + 200].On		= FALSE
		Alarm[Discharger + 200].Bag 	= 0
		Alarm[Discharger + 200].Name 	= almNoAlarm
		Alarm[Discharger + 200].Beacon	= FALSE
	ENDIF

	D[1017]		= ManualBagsRecirc

	IF ProgramRunning THEN
		D[18 + n]	= 1
	ELSE
		D[18 + n]	= 0
	ENDIF

	D32[30 + Discharger] 	= Uld[Discharger].FIFOCustomer
	;D[187 + n] 		= Uld[Discharger].FIFONextCustomer

END_PROGRAM
```

### Program Logical/Sequences/10ms/sortingBelts1 (IEC) - *Sorting Belts

#### Variables.var
```iecst
VAR CONSTANT
	LOCAL_MAX_DRIVES : USINT := 3;
END_VAR
(*Insert your comment here.*)
VAR
	beltSpeed : ARRAY[0..LOCAL_MAX_DRIVES] OF UINT;
	drive : REFERENCE TO ABB_EPL_typ;
	direction : ARRAY[0..LOCAL_MAX_DRIVES] OF ABB_DIRECTION_Enum;
	i_beltModeA : REFERENCE TO BOOL;
	i_beltModeB : REFERENCE TO BOOL;
	i_beltStart : REFERENCE TO BOOL;
	i_beltStop : REFERENCE TO BOOL;
	i_gaurdOnCentre : BOOL;
	i_gaurdOnCradle : BOOL;
	i_largeLoad : REFERENCE TO BOOL;
	i_mode : ARRAY[0..2] OF BOOL;
	i_px_beltEnd : ARRAY[0..6] OF BOOL;
	i_px_beltMid : ARRAY[0..6] OF BOOL;
	myDrive : ARRAY[0..LOCAL_MAX_DRIVES] OF USINT;
	myZone : USINT;
	n : UINT;
	nextBeltRunning : ARRAY[0..LOCAL_MAX_DRIVES] OF BOOL;
	o_lamp : ARRAY[0..2] OF BOOL;
	o_run : ARRAY[0..LOCAL_MAX_DRIVES] OF BOOL;
	runBelts : ARRAY[0..LOCAL_MAX_DRIVES] OF BOOL;
	sortingMode : USINT;
	start : ARRAY[0..2] OF F_TRIG;
	ton_LargeLoadSB6 : TON_10ms;
	ton_MergeLoadSB6 : TON_10ms;
	i_beltStart_2 : REFERENCE TO BOOL;
	i_beltStop_2 : REFERENCE TO BOOL;
	comm : REFERENCE TO Comm_typ;
	i_px_fin : ARRAY[0..6] OF BOOL;
	o_fin_up : ARRAY[0..6] OF BOOL;
	ton_fin : ARRAY[0..6] OF TON_10ms;
	linenAtFin_time : UDINT;
	ton_runSortingBelt : ARRAY[1..2] OF TOF_10ms;
	o_fin_down : ARRAY[0..6] OF BOOL;
	WasherUnloading : BOOL;
	Testwash : BOOL;
	relay : BOOL;
	ManaulOperation : BOOL;
	switch : BOOL;
	InchPushButton : BOOL;
	momentery : BOOL;
	BeltA_DetectsLargeLoad : BOOL;
	photocell : BOOL;
	A : BOOL;
	SBA_PhotocellReverse : BOOL;
	SB : BOOL;
	SBA_Photocell : BOOL;
	linen : BOOL;
	SB_3PhotocellFullBottom : BOOL;
	conveyor : BOOL;
	SB4_PhotoCell : BOOL;
	LoadOK : BOOL;
	push : BOOL;
	mySeq : INT;
	alarm : REFERENCE TO Alm;
	step : INT;
	pls : BOOL;
	lastStep : INT;
	myBag : UINT;
	O_BrakeA : BOOL;
	StopBelts : BOOL;
	O_BrakeSB3 : BOOL;
	STEP : BOOL;
	ResetBelt : BOOL;
	ResetBeltET : UDINT;
	ton_10ms_ResetBelt : TON_10ms;
	Alternate : USINT;
	PT : INT;
	ton_10ms_FDC1 : TON_10ms;
	ton_10ms_Clear : TON_10ms;
	ton_10ms_FDC2 : TON_10ms;
	ton_10ms_Clear1 : TON_10ms;
	O_BeltReadyFDC1 : BOOL;
	O_BeltReadyFDC2 : BOOL;
	O_RunBeltA_Forward : BOOL;
	RunBelt : BOOL;
	ton_10ms_StopBelts : TON_10ms;
	ton_10ms_RunBelt : TOF_10ms;
	O_RunBeltA_Slow : BOOL;
	kev : BOOL;
	O_RunBeltB_Forward : BOOL;
	O_RunBeltB_Speed2 : BOOL;
	O_Runbelt3_Forward : BOOL;
	O_RunBelt3_Speed2 : BOOL;
	LinenDetected : BOOL;
	ton_10ms_SB_3Full : TON_10ms;
	ton_10ms_SB_3Clear : TON_10ms;
	ton_10ms_LinenDetected : TON_10ms;
	SB2Clear : BOOL;
	ton_10ms_SB2Clear : TON_10ms;
	SlowA : BOOL;
	BeltAlarm : BOOL;
	ENDIF : BOOL;
	SBBeltClear : BOOL;
	ton_10ms_SBBeltClear : TON_10ms;
	AlarmLamp : BOOL;
	O_OK_Lamp : BOOL;
	O_PauseUnloading : BOOL;
	Slow1 : BOOL;
	O_RunBeltB_Slow : BOOL;
	SlowB : BOOL;
	O_Runbelt3_Slow : BOOL;
	Slow3 : BOOL;
	ton_10ms_Slow1 : TON_10ms;
	O_ReverseBeltA : BOOL;
	ton_10ms_SlowA : TON_10ms;
	ton_10ms_SlowB : TON_10ms;
	ton_10ms_Slow3 : TON_10ms;
	timerAlarm : TON_10ms;
END_VAR
```

#### Main.st
```iecst
PROGRAM _INIT
myZone 			:= 0;
//myDrive[1]		:= 1;
//myDrive[2]		:= 2;
//myDrive[3]		:= 3;
//myDrive[4]		:= 4;
//myDrive[5]		:= 5;
//myDrive[6]		:= 6;

//Comm for foul wash belt
comm							ACCESS ADR(Comm[21]);

FOR n := 1 TO LOCAL_MAX_DRIVES DO
	myDrive[n]					:= UINT_TO_USINT(n);
	drive						ACCESS ADR(ABB_EPL.Drives[myDrive[n]]);

	direction[n] 				:= ABB_DIRECTION_FWD;
	drive.Cmd.Acc_seconds := 1; //0 will default to 3 seconds
	drive.Cmd.Dec_seconds := 0.5; //0 will default to 3 second
	CASE n OF
		1:
			beltSpeed[n] 	:= 70;
			drive.Cmd.MotorSize := ABB_MOTOR_0_37KW_0_97A_1342;

		2:
			beltSpeed[n] 	:= 70;
			drive.Cmd.BrakeFitted := 1;
			drive.Cmd.MotorSize := ABB_MOTOR_0_75KW;

		3:
			beltSpeed[n] 	:= 70;
			drive.Cmd.MotorSize := ABB_MOTOR_0_25KW;

		END_CASE;
mySeq						:= 36;
alarm						ACCESS ADR(Alarm[mySeq]);

(*	i_largeLoad	ACCESS ADR(X[0].X02);	                                              SB-B           _________________________________________________
	i_beltStart ACCESS ADR(X[351].X06);	                                             |         |                                                      ]
	i_beltStop 	ACCESS ADR(X[351].X07);	                                             |         |                SB-A                                  ]
	                                                                                 |         |                                                      ]
	i_beltStart_2 ACCESS ADR(X[352].X06);  	                                         |         |     __________________________________________________
	i_beltStop_2 ACCESS ADR(X[352].X07);	                                         |         |
		                                                                             |         |
	i_beltModeA	ACCESS ADR(X[0].X01);                                                |         |
	i_beltModeB	ACCESS ADR(X[0].X02);	                                             |         |
	                                                                                 |         |
	linenAtFin_time := 500;	                                                      |         |         *)

END_FOR;

END_PROGRAM

PROGRAM _CYCLIC

alarm.Name 		:= 0;
alarm.Beacon	:= TRUE;
alarm.Extra		:= 0;
alarm.Bag		:= myBag;
alarm.Time		:= 3000;

//Setup Sequence
step := D[900 + mySeq];
//Setup Pulse contact
pls := (step <> lastStep);
lastStep := step;

sortingMode := UINT_TO_USINT(D[936]);

WasherUnloading         := X[12].X04 OR Testwash;//relay in panel signal from washers;
ManaulOperation         := X[12].X16;//switch on remote box;
InchPushButton          := X[12].X12;//momentery push button;

BeltA_DetectsLargeLoad  := X[12].X14;//photocell on belt SB-A;
SBA_PhotocellReverse    := X[12].X10;//photocell at end OF SB-A in reverse;

SBA_Photocell           := X[12].X15;//linen detected end OF SB-A;
SB_3PhotocellFullBottom := X[12].X11;//linen at end OF conveyor when reversing;

SB4_PhotoCell           := X[12].X13;

LoadOK                  := X[15].X01;//push button on panel;

Request.SB[2]           := FALSE;

IF ((step >= 3) AND (step <= 6)) OR ((step >=7) AND (step <= 10)) THEN
    O_BrakeA := TRUE;
ELSE
    O_BrakeA := FALSE;
END_IF;

IF ((step >= 4) AND (step <= 9) AND (step <> 5) AND NOT StopBelts)  THEN
    O_BrakeSB3 := TRUE;
ELSE
    O_BrakeSB3 := FALSE;
END_IF;

//;Sequence
IF (STEP = 0) THEN
	//disabled
END_IF;

ton_10ms_ResetBelt(IN:= (step = 1),PT:= 200);
//TON_10ms(((STEP = 1)),200,ResetBelt,ResetBeltET)
IF (step = 1) THEN
	IF ResetBelt THEN
		D[936] := 2;
	END_IF;
END_IF;

IF (step <> 2) THEN
	Alternate := 1;
END_IF;

//;Wait FOR unload signal AND manaul OR auto
ton_10ms_FDC1(IN:= ((step = 2)AND (Alternate = 1)),PT:= 500);        //      (((STEP = 2) AND (Alternate = 1)),500,FDC1,FDC1ET)
ton_10ms_Clear(IN:=((step = 2)AND (Alternate = 2)),PT:= 200);
ton_10ms_FDC2(IN:= ((step = 2)AND (Alternate = 3)),PT:= 500);//ton_10ms(((STEP = 2)AND (Alternate = 3)),500,FDC2,FDC2ET)
ton_10ms_Clear1(IN:=((step = 2)AND (Alternate = 4)),PT:= 200);//ton_10ms(((STEP = 2)AND (Alternate = 4)),200,Clear1,Clear1ET)

IF (step = 2) THEN
	IF ((Alternate > 4) OR (Alternate <= 0)) THEN
		 Alternate := 1;
    END_IF;

   IF ton_10ms_FDC1.Q THEN
    	Alternate := 2;
    ELSIF ton_10ms_Clear.Q THEN
    	Alternate := 3;
    ELSIF ton_10ms_FDC2.Q THEN
    	Alternate := 4;
	ELSIF ton_10ms_Clear1.Q THEN
		Alternate := 1;
	END_IF;

	O_BeltReadyFDC1 := (Alternate = 1);
    O_BeltReadyFDC2 := (Alternate = 3);

	//;O_BeltReadyFDC1 = Std.M9035
	//;O_BeltReadyFDC2 = NOT Std.M9035

	IF ((WasherUnloading = TRUE) AND (NOT ManaulOperation)) THEN
		D[936] := 4; //;changed from 3
	ELSIF ((WasherUnloading = TRUE) AND  (ManaulOperation = TRUE)) THEN
		D[936] := 10;
	END_IF;
END_IF;

//run belt at 10 meters a minute
IF (step = 3) THEN
	O_RunBeltA_Forward := TRUE; //;10ms
	IF (BeltA_DetectsLargeLoad = TRUE) THEN
		D[936] := 7;
	END_IF;
	IF (SBA_Photocell = TRUE) THEN
		D[936] := 4;
	END_IF;
END_IF;

ton_10ms_StopBelts(IN:=((step = 6) AND NOT RunBelt),PT:= 500);
ton_10ms_RunBelt(IN:=StopBelts,PT:= 500);

ton_10ms_SB_3Full(IN:=(SB_3PhotocellFullBottom = TRUE),PT:= 50);
ton_10ms_SB_3Clear(IN:=(SB_3PhotocellFullBottom = FALSE),PT:= 50);
ton_10ms_LinenDetected(IN:=((step = 4) AND SB4_PhotoCell),PT:= 600);
IF (step = 4) THEN

	     O_RunBeltA_Forward   := TRUE; //;SB_3Clear
	     O_RunBeltA_Slow      := kev;
	     O_RunBeltB_Forward   := TRUE;
	     O_RunBeltB_Speed2    := TRUE;
	     O_Runbelt3_Forward   := TRUE;
	     O_RunBelt3_Speed2    := TRUE;

	IF (BeltA_DetectsLargeLoad = TRUE) THEN
		D[936] := 8;
	END_IF;
	IF (LinenDetected = TRUE) THEN
		D[936] := 5;
	END_IF;
END_IF;

//I_SafetyRelayOn AND sb2 NOT running
ton_10ms_SB2Clear(IN:=(NOT Std.HaltSys AND (Y[14].Y04= TRUE) AND NOT Y[14].Y03),PT:= 1700);
IF (step = 5) THEN
	Request.SB[2] := TRUE;
	IF (ton_10ms_SB2Clear.Q = TRUE) THEN
		D[936] := 6;
	END_IF;
END_IF;

//;run belts at 10ms
ton_10ms_SBBeltClear(IN:=((step = 6) AND (NOT SB4_PhotoCell) AND (NOT Std.HaltSys = TRUE)),PT:= 3000);
IF (step = 6) THEN
		Request.SB[2] := TRUE;
    IF ((Y[14].Y04 = TRUE) AND NOT StopBelts) THEN
		 O_RunBeltA_Forward         := TRUE;
		 O_RunBeltA_Slow            := SlowA;
		 O_RunBeltB_Forward         := TRUE;
		 O_Runbelt3_Forward         := TRUE;
	END_IF;
	IF (BeltA_DetectsLargeLoad = TRUE) THEN
		BeltAlarm   := TRUE;
		D[936] := 9;
	END_IF;
	IF SBBeltClear THEN
		D[936] := 1;
	END_IF;
END_IF;

//;Large load from step 3
IF (step = 7) THEN
	AlarmLamp              := TRUE;
	O_OK_Lamp              := TRUE;
	O_PauseUnloading       := TRUE;
	IF (InchPushButton AND (SB4_PhotoCell = FALSE)) THEN
	    O_RunBeltA_Forward := TRUE;

		O_RunBeltA_Slow    := ton_10ms_Slow1.Q;

	END_IF;
	IF LoadOK THEN
		D[936] := 3;
	END_IF;
END_IF;

ton_10ms_Slow1(IN:=(O_RunBeltA_Forward = TRUE),PT:= 50);

//;Large load from step 4
IF (step = 8) THEN
	AlarmLamp              := TRUE;
	O_OK_Lamp              := TRUE;
	O_PauseUnloading       := TRUE;
	IF (InchPushButton AND (SB4_PhotoCell = FALSE)) THEN
	    O_RunBeltA_Forward := TRUE;
	    O_RunBeltA_Slow    := SlowA;
	    O_RunBeltB_Forward := TRUE;
	    O_RunBeltB_Slow    := SlowB;
	    O_Runbelt3_Forward := TRUE;
	    O_Runbelt3_Slow    := Slow3;

	END_IF;
	IF LoadOK THEN
		D[936] := 4;
	END_IF;
  END_IF;

//;Large load from step 6
IF (step = 9) THEN
	AlarmLamp              := TRUE;
	O_OK_Lamp              := TRUE;
	O_PauseUnloading       := TRUE;
	IF (InchPushButton AND (SB4_PhotoCell = FALSE)) THEN
		O_RunBeltA_Slow    := SlowA;
	    O_RunBeltA_Forward := TRUE;
	    O_RunBeltB_Forward := TRUE;
	    O_RunBeltB_Slow    := SlowB;
	    O_Runbelt3_Forward := TRUE;
	    O_Runbelt3_Slow    := Slow3;

	END_IF
	IF LoadOK THEN
		D[936] := 6;
	END_IF
END_IF

//;manual mode
IF (step = 10) THEN
//	;AlarmLamp              = TRUE
	O_OK_Lamp              := TRUE;
//	;O_PauseUnloading       := TRUE;
	IF (InchPushButton  AND (SBA_PhotocellReverse = FALSE)) THEN
	    O_ReverseBeltA    := TRUE;
	END_IF;
	IF LoadOK THEN
		D[936] := 1;
	END_IF;
END_IF;

//Alarms
timerAlarm(IN := NOT pls AND (alarm.Name > 0),PT:= alarm.Time);

alarm.On 	:= timerAlarm.Q;
alarm.ET 	:= timerAlarm.ET;

ton_10ms_SlowA(IN:=(O_RunBeltA_Forward = TRUE),PT:= 50);
ton_10ms_SlowB(IN:=(O_RunBeltB_Forward = TRUE),PT:= 50);
ton_10ms_Slow3(IN:=(O_Runbelt3_Forward = TRUE),PT:= 50);

//;Outputs
Y[12].Y15 := AlarmLamp;// ;YC15
Y[15].Y01 := O_OK_Lamp;// ;Lamp on push button box YF01
Y[12].Y14  := O_BeltReadyFDC1;//;YC14
Y[12].Y16  := O_BeltReadyFDC2;//;YC16

Y[14].Y13  := O_RunBeltA_Slow;// ;YE13
Y[14].Y09 := O_RunBeltA_Forward;//;YE09

Y[14].Y11 := O_RunBeltB_Forward;//;YE11

Y[14].Y05 := O_Runbelt3_Forward;//  ;YYE05

Y[14].Y12 := O_RunBeltB_Slow;//;YE12

Y[14].Y08 := O_Runbelt3_Slow;// ;YE08

Y[14].Y10 := O_ReverseBeltA;//    ;YE10

Y[15].Y02 := O_RunBeltB_Speed2;// ;YF02

Y[15].Y03 := O_RunBelt3_Speed2;// ;YF03

Y[15].Y04 := O_PauseUnloading;//  ;YF04

Y[14].Y06 := Y[14].Y05;

Y[14].Y16 := O_BrakeA;// ;YE16
Y[14].Y14 := O_BrakeSB3;//  ;YE14

CASE sortingMode OF

	99: //Test Mode

		runBelts[1] := (D[2] > 0);
		runBelts[2] := (D[3] > 0);
		runBelts[3] := (D[4] > 0);

END_CASE;

FOR n := 1 TO LOCAL_MAX_DRIVES DO

	drive						ACCESS ADR(ABB_EPL.Drives[myDrive[n]]);
//	IF (ABB_EPL.Settings[n].Fast > 0) THEN
//		beltSpeed[n] := ABB_EPL.Settings[n].Fast;
//	END_IF;

	drive.Cmd.TargetVelocity := beltSpeed[n];
	drive.Cmd.Run := o_run[n] AND NOT Std.HaltSysZone[myZone];
	drive.Cmd.QuickStop 	:= NOT Std.HaltSysZone[myZone];
	drive.Cmd.Direction		:= direction[n];
	Indication[12 + n] 		:= drive.Status.Running;
END_FOR;

END_PROGRAM
```

### Package Logical/Sequences/200ms - 200ms Tasks

### Package Logical/Sequences/200ms/CAN - CAN Communication Variables

### CAN.var
```iecst
VAR
	CAN : ARRAY[0..32] OF CAN_Vars;
END_VAR
VAR CONSTANT
	MAX_COMM : USINT := 25;
END_VAR
VAR
	Comm : ARRAY[0..MAX_COMM] OF Comm_typ;
END_VAR
```
